KUKA KRL program: MyProgram_086().src

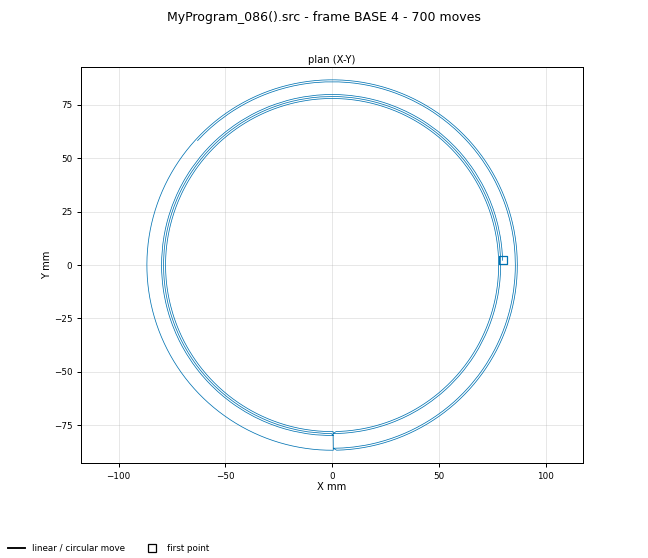
[picture p0: tool path of MyProgram_086().src in frame BASE 4, 700 of 700 moves have a stored position in this frame; points joined in program order, loops and branches not executed]
&ACCESS RVP
&REL 1
&PARAM TEMPLATE = C:\KRC\Roboter\Template\vorgabe
&PARAM EDITMASK = *
DEF MyProgram_086()
; ---- Setting reference (Base) ----
$BASE = BASE_DATA[4]

; --------------------------
; ---- Setting tool (TCP) ----
$TOOL = TOOL_DATA[3]
; --------------------------

$VEL.CP = VEL_APROX_PRINT
Startdeposition()
$VEL.CP = VEL_PRINT
LIN {X 79.8742,Y 2.2154,Z 84,A -3.1634,B 24.9021,C -2.2842,E1 25.1597,E2 447.7459} C_DIS
LIN {X 79.7565,Y 4.8855,Z 84,A -1.5386,B 24.9024,C -2.2808,E1 25.1594,E2 446.1387} C_DIS
LIN {X 79.546,Y 7.5648,Z 84,A 0.5064,B 24.9016,C -2.2907,E1 25.1589,E2 444.0824} C_DIS
LIN {X 79.2109,Y 10.5084,Z 84,A 2.7603,B 24.9006,C -2.3016,E1 25.1581,E2 441.8162} C_DIS
LIN {X 78.7938,Y 13.2771,Z 84,A 4.7205,B 24.9002,C -2.3063,E1 25.1573,E2 439.8564} C_DIS
LIN {X 77.6208,Y 18.9672,Z 84,A 8.4482,B 24.9003,C -2.305,E1 25.1551,E2 436.1534} C_DIS
LIN {X 76.3858,Y 23.452,Z 84,A 12.1024,B 24.8986,C -2.3252,E1 25.1523,E2 432.4725} C_DIS
LIN {X 75.4106,Y 26.4193,Z 84,A 14.3588,B 24.8979,C -2.3323,E1 25.1503,E2 430.2119} C_DIS
LIN {X 74.0231,Y 30.0886,Z 84,A 17.0668,B 24.8975,C -2.3371,E1 25.1475,E2 427.5076} C_DIS
LIN {X 72.6892,Y 33.1839,Z 84,A 19.5229,B 24.8968,C -2.3452,E1 25.1448,E2 425.0459} C_DIS
LIN {X 71.424,Y 35.8258,Z 84,A 21.7203,B 24.896,C -2.3541,E1 25.142,E2 422.8392} C_DIS
LIN {X 70.1389,Y 38.2794,Z 84,A 23.7,B 24.8956,C -2.3593,E1 25.1394,E2 420.8576} C_DIS
LIN {X 67.1297,Y 43.3403,Z 84,A 27.8834,B 24.8947,C -2.3691,E1 25.1333,E2 416.6724} C_DIS
LIN {X 65.2345,Y 46.1444,Z 84,A 30.2162,B 24.8944,C -2.3722,E1 25.1296,E2 414.3437} C_DIS
LIN {X 62.1422,Y 50.2304,Z 84,A 33.417,B 24.8949,C -2.3662,E1 25.1243,E2 411.1722} C_DIS
LIN {X 59.7766,Y 53.0248,Z 84,A 37.0655,B 24.8915,C -2.4041,E1 25.1174,E2 407.4506} C_DIS
LIN {X 57.5676,Y 55.4135,Z 84,A 39.0218,B 24.8921,C -2.3974,E1 25.1137,E2 405.5186} C_DIS
LIN {X 54.5308,Y 58.4041,Z 84,A 42.8995,B 24.8893,C -2.4292,E1 25.1057,E2 401.5814} C_DIS
LIN {X 50.973,Y 61.5346,Z 84,A 44.8682,B 24.8927,C -2.3915,E1 25.1017,E2 399.7098} C_DIS
LIN {X 49.2422,Y 62.9293,Z 84,A 46.8182,B 24.8914,C -2.4053,E1 25.0974,E2 397.7345} C_DIS
LIN {X 44.8304,Y 66.1436,Z 84,A 50.2204,B 24.8922,C -2.3963,E1 25.0898,E2 394.3654} C_DIS
LIN {X 42.7835,Y 67.4871,Z 84,A 52.2562,B 24.8912,C -2.4075,E1 25.085,E2 392.3098} C_DIS
LIN {X 40.8002,Y 68.703,Z 84,A 54.7814,B 24.8886,C -2.436,E1 25.0788,E2 389.7249} C_DIS
LIN {X 37.7018,Y 70.4522,Z 84,A 56.7061,B 24.8901,C -2.4204,E1 25.0741,E2 387.8427} C_DIS
LIN {X 34.3391,Y 72.1502,Z 84,A 59.5121,B 24.8895,C -2.4269,E1 25.0671,E2 385.0287} C_DIS
LIN {X 30.3149,Y 73.931,Z 84,A 62.4788,B 24.8897,C -2.4246,E1 25.0595,E2 382.0745} C_DIS
LIN {X 26.5785,Y 75.3548,Z 84,A 64.9595,B 24.8905,C -2.4159,E1 25.0531,E2 379.6198} C_DIS
LIN {X 24.1474,Y 76.17,Z 84,A 67.3413,B 24.8889,C -2.4333,E1 25.0467,E2 377.2012} C_DIS
LIN {X 21.1695,Y 77.05,Z 84,A 69.6421,B 24.8885,C -2.437,E1 25.0405,E2 374.8954} C_DIS
LIN {X 17.4919,Y 77.9679,Z 84,A 72.8738,B 24.887,C -2.4535,E1 25.0316,E2 371.6289} C_DIS
LIN {X 13.8906,Y 78.6883,Z 84,A 74.367,B 24.89,C -2.4213,E1 25.0277,E2 370.2138} C_DIS
LIN {X 8.6493,Y 79.4357,Z 84,A 78.2763,B 24.8896,C -2.4254,E1 25.0169,E2 366.2982} C_DIS
LIN {X 3.806,Y 79.8147,Z 84,A 82.6374,B 24.8873,C -2.4507,E1 25.0046,E2 361.8791} C_DIS
LIN {X 0.5734,Y 79.9025,Z 84,A 84.7785,B 24.8878,C -2.4452,E1 24.9986,E2 359.7512} C_DIS
LIN {X -3.1784,Y 79.8417,Z 84,A 87.9123,B 24.8867,C -2.457,E1 24.9898,E2 356.5887} C_DIS
LIN {X -7.2148,Y 79.5783,Z 84,A 89.9291,B 24.8891,C -2.4306,E1 24.9844,E2 354.6338} C_DIS
LIN {X -13.3811,Y 78.7764,Z 84,A 95.4024,B 24.8868,C -2.4562,E1 24.9691,E2 349.0949} C_DIS
LIN {X -17.7165,Y 77.9162,Z 84,A 97.6435,B 24.8894,C -2.4274,E1 24.9631,E2 346.9195} C_DIS
LIN {X -20.8905,Y 77.1254,Z 84,A 100.0246,B 24.8895,C -2.4261,E1 24.9567,E2 344.5381} C_DIS
LIN {X -26.7737,Y 75.2863,Z 84,A 104.5281,B 24.8898,C -2.4232,E1 24.9447,E2 340.0333} C_DIS
LIN {X -30.0238,Y 74.0495,Z 84,A 107.3916,B 24.8892,C -2.4299,E1 24.9372,E2 337.1475} C_DIS
LIN {X -34.5431,Y 72.0522,Z 84,A 110.4827,B 24.8908,C -2.4123,E1 24.9295,E2 334.0908} C_DIS
LIN {X -37.6093,Y 70.5015,Z 84,A 113.0625,B 24.8908,C -2.4113,E1 24.9231,E2 331.5062} C_DIS
LIN {X -42.7396,Y 67.5136,Z 84,A 117.0511,B 24.8922,C -2.3965,E1 24.9136,E2 327.5408} C_DIS
LIN {X -45.878,Y 65.421,Z 84,A 120.3122,B 24.8914,C -2.406,E1 24.906,E2 324.246} C_DIS
LIN {X -49.9813,Y 62.3441,Z 84,A 124.1225,B 24.8918,C -2.4017,E1 24.8976,E2 320.4319} C_DIS
LIN {X -52.7972,Y 59.9774,Z 84,A 126.8256,B 24.8921,C -2.3975,E1 24.8919,E2 317.7282} C_DIS
LIN {X -55.1723,Y 57.8006,Z 84,A 128.6467,B 24.8938,C -2.3792,E1 24.8883,E2 315.9432} C_DIS
LIN {X -57.5075,Y 55.4763,Z 84,A 131.6065,B 24.8929,C -2.3893,E1 24.8824,E2 312.9468} C_DIS
LIN {X -59.8884,Y 52.8992,Z 84,A 133.2739,B 24.8954,C -2.3607,E1 24.8795,E2 311.3401} C_DIS
LIN {X -61.9095,Y 50.5175,Z 84,A 135.7729,B 24.8954,C -2.3617,E1 24.875,E2 308.8273} C_DIS
LIN {X -65.6702,Y 45.5207,Z 84,A 140.2241,B 24.8965,C -2.3488,E1 24.8676,E2 304.3853} C_DIS
LIN {X -67.0145,Y 43.5198,Z 84,A 142.3289,B 24.896,C -2.3537,E1 24.8644,E2 302.2582} C_DIS
LIN {X -69.2019,Y 39.9481,Z 84,A 144.8295,B 24.8979,C -2.3322,E1 24.8608,E2 299.796} C_DIS
LIN {X -71.2813,Y 36.1081,Z 84,A 147.7071,B 24.8993,C -2.3167,E1 24.8571,E2 296.9403} C_DIS
LIN {X -72.814,Y 32.9069,Z 84,A 150.6411,B 24.8991,C -2.319,E1 24.8535,E2 293.9847} C_DIS
LIN {X -74.8991,Y 27.8408,Z 84,A 154.4993,B 24.9003,C -2.3053,E1 24.8495,E2 290.1378} C_DIS
LIN {X -76.4902,Y 23.1115,Z 84,A 158.2746,B 24.9008,C -2.2992,E1 24.8462,E2 286.3553} C_DIS
LIN {X -77.3182,Y 20.167,Z 84,A 160.5268,B 24.9013,C -2.2939,E1 24.8446,E2 284.1028} C_DIS
LIN {X -78.0736,Y 17.0075,Z 84,A 162.8457,B 24.9019,C -2.2863,E1 24.8431,E2 281.7885} C_DIS
LIN {X -78.7311,Y 13.6505,Z 84,A 166.1222,B 24.9008,C -2.2996,E1 24.8415,E2 278.4606} C_DIS
LIN {X -79.3072,Y 9.763,Z 84,A 168.4445,B 24.9027,C -2.2779,E1 24.8407,E2 276.1764} C_DIS
LIN {X -79.8336,Y 3.3663,Z 84,A 173.7794,B 24.9023,C -2.2821,E1 24.8398,E2 270.7993} C_DIS
LIN {X -79.8974,Y -1.1225,Z 84,A 175.7486,B 24.9059,C -2.2397,E1 24.8398,E2 268.9195} C_DIS
LIN {X -79.8317,Y -3.4108,Z 84,A 177.6251,B 24.9059,C -2.2405,E1 24.84,E2 267.0298} C_DIS
LIN {X -79.4763,Y -8.2616,Z 84,A -178.2229,B 24.9053,C -2.2466,E1 24.841,E2 262.8384} C_DIS
LIN {X -79.0723,Y -11.5061,Z 84,A -176.628,B 24.9076,C -2.22,E1 24.8416,E2 261.2975} C_DIS
LIN {X -78.6483,Y -14.113,Z 84,A -173.8348,B 24.9061,C -2.2373,E1 24.843,E2 258.4465} C_DIS
LIN {X -77.9265,Y -17.6722,Z 84,A -172.049,B 24.9085,C -2.2081,E1 24.844,E2 256.7197} C_DIS
LIN {X -77.2337,Y -20.4894,Z 84,A -169.8346,B 24.9088,C -2.2053,E1 24.8456,E2 254.4992} C_DIS
LIN {X -76.4721,Y -23.1726,Z 84,A -167.7993,B 24.9092,C -2.2002,E1 24.8472,E2 252.4643} C_DIS
LIN {X -75.6471,Y -25.7351,Z 84,A -165.9949,B 24.9099,C -2.1913,E1 24.8487,E2 250.6709} C_DIS
LIN {X -74.8294,Y -28.0247,Z 84,A -164.0957,B 24.91,C -2.1902,E1 24.8506,E2 248.7635} C_DIS
LIN {X -73.1802,Y -32.0845,Z 84,A -160.7297,B 24.9103,C -2.1871,E1 24.8542,E2 245.3863} C_DIS
LIN {X -71.665,Y -35.3396,Z 84,A -158.3657,B 24.9113,C -2.1744,E1 24.8571,E2 243.0397} C_DIS
LIN {X -70.2189,Y -38.132,Z 84,A -155.2566,B 24.91,C -2.1908,E1 24.8613,E2 239.8751} C_DIS
LIN {X -68.2289,Y -41.5881,Z 84,A -153.7955,B 24.9136,C -2.1466,E1 24.8632,E2 238.5119} C_DIS
LIN {X -65.3218,Y -46.022,Z 84,A -149.2606,B 24.9128,C -2.1561,E1 24.8703,E2 233.9316} C_DIS
LIN {X -63.2139,Y -48.8748,Z 84,A -146.7523,B 24.9134,C -2.149,E1 24.8745,E2 231.4282} C_DIS
LIN {X -61.0851,Y -51.5123,Z 84,A -143.5632,B 24.9122,C -2.1637,E1 24.8803,E2 228.1893} C_DIS
LIN {X -58.459,Y -54.474,Z 84,A -141.8,B 24.915,C -2.1287,E1 24.8835,E2 226.502} C_DIS
LIN {X -56.8071,Y -56.1934,Z 84,A -138.8409,B 24.9126,C -2.1587,E1 24.8895,E2 223.4585} C_DIS
LIN {X -53.5902,Y -59.2704,Z 84,A -136.8565,B 24.9157,C -2.1196,E1 24.8934,E2 221.5593} C_DIS
LIN {X -50.8929,Y -61.6012,Z 84,A -133.9567,B 24.9154,C -2.1241,E1 24.8996,E2 218.6378} C_DIS
LIN {X -47.3833,Y -64.3398,Z 84,A -131.2008,B 24.9168,C -2.1066,E1 24.9056,E2 215.9134} C_DIS
LIN {X -45.2583,Y -65.8529,Z 84,A -129.046,B 24.9164,C -2.1112,E1 24.9106,E2 213.7403} C_DIS
LIN {X -40.5803,Y -68.833,Z 84,A -125.0904,B 24.9169,C -2.1046,E1 24.92,E2 209.7878} C_DIS
LIN {X -36.4922,Y -71.085,Z 84,A -121.1636,B 24.916,C -2.1164,E1 24.9297,E2 205.8221} C_DIS
LIN {X -32.4299,Y -73.029,Z 84,A -117.9364,B 24.9163,C -2.1127,E1 24.9379,E2 202.5957} C_DIS
LIN {X -28.8497,Y -74.5157,Z 84,A -115.4468,B 24.9172,C -2.1018,E1 24.9443,E2 200.1266} C_DIS
LIN {X -25.242,Y -75.8134,Z 84,A -112.9215,B 24.9178,C -2.0932,E1 24.9509,E2 197.6168} C_DIS
LIN {X -22.0228,Y -76.8101,Z 84,A -110.403,B 24.9178,C -2.0944,E1 24.9577,E2 195.0912} C_DIS
LIN {X -18.1488,Y -77.8164,Z 84,A -107.4559,B 24.9177,C -2.095,E1 24.9657,E2 192.1384} C_DIS
LIN {X -11.9311,Y -79.0093,Z 84,A -103.2308,B 24.9185,C -2.0844,E1 24.9773,E2 187.9342} C_DIS
LIN {X -7.865,Y -79.5178,Z 84,A -100.2852,B 24.9185,C -2.0841,E1 24.9854,E2 184.9873} C_DIS
LIN {X -1.223,Y -79.8956,Z 84,A -95.4367,B 24.9183,C -2.0867,E1 24.9989,E2 180.1315} C_DIS
LIN {X 0.4916,Y -79.9011,Z 84,A -94.4036,B 24.9188,C -2.0813,E1 25.0018,E2 179.1113} C_DIS
Enddeposition()
LIN {X 0.4916,Y -79.9011,Z 84,A -94.4036,B 24.9188,C -2.0813,E1 25.0018,E2 179.1113} C_DIS
Startdeposition()
$VEL.CP = VEL_PRINT
LIN {X -0.3135,Y -78.968,Z 84,A -95.3503,B 24.9183,C -2.0869,E1 24.9992,E2 180.0445} C_DIS
LIN {X -3.6516,Y -78.8844,Z 84,A -98.627,B 24.9202,C -2.0625,E1 24.9899,E2 183.3797} C_DIS
LIN {X -11.2534,Y -78.1626,Z 84,A -103.0469,B 24.9177,C -2.0945,E1 24.9778,E2 187.7261} C_DIS
LIN {X -14.5877,Y -77.6101,Z 84,A -106.1891,B 24.9192,C -2.076,E1 24.969,E2 190.9155} C_DIS
LIN {X -16.7787,Y -77.1653,Z 84,A -108.0748,B 24.9197,C -2.0694,E1 24.9638,E2 192.819} C_DIS
LIN {X -20.6747,Y -76.214,Z 84,A -110.5178,B 24.9186,C -2.0839,E1 24.9573,E2 195.2311} C_DIS
LIN {X -22.947,Y -75.5622,Z 84,A -112.4428,B 24.9189,C -2.0793,E1 24.9521,E2 197.1703} C_DIS
LIN {X -25.8684,Y -74.6118,Z 84,A -114.6287,B 24.9187,C -2.0823,E1 24.9463,E2 199.3533} C_DIS
LIN {X -28.9712,Y -73.4622,Z 84,A -116.9095,B 24.9183,C -2.0878,E1 24.9404,E2 201.6258} C_DIS
LIN {X -32.0325,Y -72.1812,Z 84,A -119.3726,B 24.9182,C -2.0888,E1 24.9341,E2 204.0923} C_DIS
LIN {X -36.2142,Y -70.1757,Z 84,A -122.7661,B 24.9179,C -2.092,E1 24.9256,E2 207.4869} C_DIS
LIN {X -38.7437,Y -68.8114,Z 84,A -124.941,B 24.9179,C -2.0924,E1 24.9202,E2 209.667} C_DIS
LIN {X -41.5484,Y -67.1555,Z 84,A -126.977,B 24.9169,C -2.1046,E1 24.9154,E2 211.6804} C_DIS
LIN {X -43.8056,Y -65.7057,Z 84,A -129.2439,B 24.9174,C -2.0991,E1 24.9101,E2 213.9678} C_DIS
LIN {X -46.2466,Y -64.0116,Z 84,A -131.5956,B 24.9174,C -2.0975,E1 24.9047,E2 216.3313} C_DIS
LIN {X -49.3608,Y -61.642,Z 84,A -134.3541,B 24.9169,C -2.1047,E1 24.8986,E2 219.0829} C_DIS
LIN {X -51.9456,Y -59.4782,Z 84,A -136.6683,B 24.9163,C -2.1128,E1 24.8937,E2 221.3868} C_DIS
LIN {X -55.1934,Y -56.479,Z 84,A -139.9523,B 24.9159,C -2.1172,E1 24.8871,E2 224.6735} C_DIS
LIN {X -57.4405,Y -54.1905,Z 84,A -142.1633,B 24.9153,C -2.1252,E1 24.8828,E2 226.8751} C_DIS
LIN {X -59.8164,Y -51.5579,Z 84,A -144.8824,B 24.9151,C -2.1272,E1 24.8777,E2 229.6016} C_DIS
LIN {X -61.7506,Y -49.2238,Z 84,A -147.0713,B 24.9147,C -2.1326,E1 24.8739,E2 231.7878} C_DIS
LIN {X -63.6304,Y -46.7676,Z 84,A -149.2643,B 24.9142,C -2.1393,E1 24.8702,E2 233.9753} C_DIS
LIN {X -65.5292,Y -44.0681,Z 84,A -151.9051,B 24.9142,C -2.1391,E1 24.866,E2 236.6298} C_DIS
LIN {X -67.2981,Y -41.3171,Z 84,A -154.3464,B 24.9138,C -2.1435,E1 24.8624,E2 239.073} C_DIS
LIN {X -69.2715,Y -37.9152,Z 84,A -157.009,B 24.9128,C -2.1559,E1 24.8588,E2 241.72} C_DIS
LIN {X -70.7826,Y -35.012,Z 84,A -159.234,B 24.912,C -2.1662,E1 24.856,E2 243.9324} C_DIS
LIN {X -71.8479,Y -32.7722,Z 84,A -161.2121,B 24.912,C -2.1667,E1 24.8536,E2 245.92} C_DIS
LIN {X -73.5353,Y -28.7848,Z 84,A -164.4106,B 24.9113,C -2.1743,E1 24.8502,E2 249.1182} C_DIS
LIN {X -74.5845,Y -25.9463,Z 84,A -166.5469,B 24.9107,C -2.1822,E1 24.8482,E2 251.2478} C_DIS
LIN {X -75.5729,Y -22.9122,Z 84,A -168.9534,B 24.9103,C -2.1868,E1 24.8462,E2 253.6571} C_DIS
LIN {X -76.4644,Y -19.7285,Z 84,A -171.3517,B 24.9097,C -2.194,E1 24.8445,E2 256.052} C_DIS
LIN {X -77.032,Y -17.3852,Z 84,A -173.1734,B 24.9094,C -2.1976,E1 24.8433,E2 257.876} C_DIS
LIN {X -77.6747,Y -14.2379,Z 84,A -175.4862,B 24.9088,C -2.2052,E1 24.8421,E2 260.1842} C_DIS
LIN {X -78.2546,Y -10.6035,Z 84,A -178.1615,B 24.9081,C -2.2134,E1 24.841,E2 262.8559} C_DIS
LIN {X -78.6457,Y -7.1324,Z 84,A 179.4961,B 24.907,C -2.2261,E1 24.8403,E2 265.1819} C_DIS
LIN {X -78.8628,Y -4.0917,Z 84,A 177.1919,B 24.9066,C -2.2308,E1 24.8399,E2 267.4887} C_DIS
LIN {X -78.9651,Y -0.824,Z 84,A 174.8111,B 24.906,C -2.2381,E1 24.8398,E2 269.8665} C_DIS
LIN {X -78.9261,Y 2.5905,Z 84,A 172.4096,B 24.9052,C -2.2479,E1 24.8399,E2 272.259} C_DIS
LIN {X -78.6598,Y 6.9801,Z 84,A 169.0099,B 24.9048,C -2.2529,E1 24.8406,E2 275.6672} C_DIS
LIN {X -78.3239,Y 10.0692,Z 84,A 167.0162,B 24.9036,C -2.2665,E1 24.8412,E2 277.6404} C_DIS
LIN {X -77.8867,Y 13.026,Z 84,A 164.5681,B 24.9036,C -2.2665,E1 24.8422,E2 280.103} C_DIS
LIN {X -77.2923,Y 16.1864,Z 84,A 162.2629,B 24.9029,C -2.2746,E1 24.8435,E2 282.4026} C_DIS
LIN {X -76.618,Y 19.1276,Z 84,A 160.0282,B 24.9024,C -2.2804,E1 24.8449,E2 284.6366} C_DIS
LIN {X -75.8653,Y 21.9234,Z 84,A 157.8612,B 24.902,C -2.2853,E1 24.8466,E2 286.8045} C_DIS
LIN {X -75.0425,Y 24.5909,Z 84,A 155.6032,B 24.902,C -2.2859,E1 24.8485,E2 289.074} C_DIS
LIN {X -74.0216,Y 27.5146,Z 84,A 153.3477,B 24.9014,C -2.2925,E1 24.8507,E2 291.3264} C_DIS
LIN {X -72.6949,Y 30.8463,Z 84,A 151.0391,B 24.9001,C -2.3076,E1 24.8531,E2 293.6119} C_DIS
LIN {X -71.5223,Y 33.4752,Z 84,A 148.9221,B 24.8996,C -2.3131,E1 24.8556,E2 295.7273} C_DIS
LIN {X -70.2745,Y 36.021,Z 84,A 146.7527,B 24.8993,C -2.3164,E1 24.8583,E2 297.9005} C_DIS
LIN {X -68.1719,Y 39.859,Z 84,A 142.8838,B 24.9,C -2.3084,E1 24.8637,E2 301.8086} C_DIS
LIN {X -66.2415,Y 42.9911,Z 84,A 140.8879,B 24.8979,C -2.3324,E1 24.8666,E2 303.7573} C_DIS
LIN {X -63.7565,Y 46.5953,Z 84,A 137.3263,B 24.898,C -2.3315,E1 24.8724,E2 307.3386} C_DIS
LIN {X -61.1955,Y 49.9117,Z 84,A 134.8544,B 24.8961,C -2.3536,E1 24.8766,E2 309.7693} C_DIS
LIN {X -59.3682,Y 52.0716,Z 84,A 132.3649,B 24.8966,C -2.3479,E1 24.8812,E2 312.2837} C_DIS
LIN {X -56.6731,Y 54.993,Z 84,A 129.6752,B 24.8955,C -2.3598,E1 24.8863,E2 314.9567} C_DIS
LIN {X -54.3673,Y 57.2742,Z 84,A 127.3959,B 24.8948,C -2.3673,E1 24.8909,E2 317.2278} C_DIS
LIN {X -52.2189,Y 59.2396,Z 84,A 125.4995,B 24.8939,C -2.3776,E1 24.8948,E2 319.1072} C_DIS
LIN {X -50.0739,Y 61.0639,Z 84,A 123.0109,B 24.8945,C -2.3707,E1 24.9002,E2 321.6217} C_DIS
LIN {X -47.3137,Y 63.2253,Z 84,A 120.4553,B 24.8941,C -2.3757,E1 24.9058,E2 324.1746} C_DIS
LIN {X -43.7728,Y 65.7273,Z 84,A 117.6723,B 24.8927,C -2.3912,E1 24.9121,E2 326.9301} C_DIS
LIN {X -41.9961,Y 66.8755,Z 84,A 115.8451,B 24.8931,C -2.3866,E1 24.9165,E2 328.7742} C_DIS
LIN {X -39.1445,Y 68.584,Z 84,A 113.6552,B 24.8922,C -2.3966,E1 24.9217,E2 330.9469} C_DIS
LIN {X -36.3929,Y 70.0841,Z 84,A 111.0691,B 24.8926,C -2.3923,E1 24.9281,E2 333.5505} C_DIS
LIN {X -33.2515,Y 71.6265,Z 84,A 108.7755,B 24.8917,C -2.4026,E1 24.9339,E2 335.8253} C_DIS
LIN {X -30.9833,Y 72.6372,Z 84,A 106.8361,B 24.8917,C -2.4016,E1 24.9388,E2 337.7716} C_DIS
LIN {X -28.0442,Y 73.821,Z 84,A 104.5278,B 24.8915,C -2.4045,E1 24.9448,E2 340.0781} C_DIS
LIN {X -23.7017,Y 75.3282,Z 84,A 101.3146,B 24.8908,C -2.4117,E1 24.9533,E2 343.2802} C_DIS
LIN {X -21.3793,Y 76.0195,Z 84,A 99.5364,B 24.8908,C -2.413,E1 24.9581,E2 345.0581} C_DIS
LIN {X -18.6628,Y 76.7314,Z 84,A 97.5178,B 24.8905,C -2.4155,E1 24.9635,E2 347.0737} C_DIS
LIN {X -15.2375,Y 77.485,Z 84,A 94.6051,B 24.8912,C -2.4078,E1 24.9716,E2 350.0082} C_DIS
LIN {X -9.5718,Y 78.3869,Z 84,A 90.7353,B 24.8902,C -2.4184,E1 24.9822,E2 353.8559} C_DIS
LIN {X -5.4515,Y 78.7801,Z 84,A 87.2166,B 24.8914,C -2.4058,E1 24.9921,E2 357.4063} C_DIS
LIN {X 1.31,Y 78.9577,Z 84,A 82.7899,B 24.8901,C -2.4202,E1 25.0043,E2 361.799} C_DIS
LIN {X 4.1367,Y 78.8603,Z 84,A 80.2315,B 24.8913,C -2.4063,E1 25.0116,E2 364.3896} C_DIS
LIN {X 8.9308,Y 78.4622,Z 84,A 77.2015,B 24.8902,C -2.4187,E1 25.0199,E2 367.3884} C_DIS
LIN {X 12.1275,Y 78.0316,Z 84,A 74.8413,B 24.8903,C -2.4175,E1 25.0264,E2 369.7491} C_DIS
LIN {X 16.3395,Y 77.2609,Z 84,A 71.7711,B 24.8903,C -2.4172,E1 25.0348,E2 372.8164} C_DIS
LIN {X 18.9682,Y 76.6569,Z 84,A 69.9746,B 24.89,C -2.4207,E1 25.0397,E2 374.6021} C_DIS
LIN {X 21.5611,Y 75.968,Z 84,A 67.8747,B 24.8905,C -2.4151,E1 25.0454,E2 376.712} C_DIS
LIN {X 24.6184,Y 75.0337,Z 84,A 65.4826,B 24.8909,C -2.4112,E1 25.0517,E2 379.1088} C_DIS
LIN {X 26.8794,Y 74.2532,Z 84,A 63.8944,B 24.8906,C -2.4139,E1 25.0559,E2 380.6874} C_DIS
LIN {X 29.5861,Y 73.2169,Z 84,A 61.0395,B 24.8928,C -2.3903,E1 25.0634,E2 383.5919} C_DIS
LIN {X 32.9059,Y 71.7873,Z 84,A 58.8986,B 24.8918,C -2.4011,E1 25.0688,E2 385.7018} C_DIS
LIN {X 36.3828,Y 70.0893,Z 84,A 56.1972,B 24.8918,C -2.4006,E1 25.0755,E2 388.3969} C_DIS
LIN {X 40.1048,Y 68.0266,Z 84,A 53.2732,B 24.8918,C -2.4011,E1 25.0826,E2 391.3111} C_DIS
LIN {X 42.6665,Y 66.4498,Z 84,A 51.0113,B 24.8923,C -2.3955,E1 25.0879,E2 393.5792} C_DIS
LIN {X 45.8019,Y 64.3289,Z 84,A 48.4166,B 24.8923,C -2.3955,E1 25.0939,E2 396.165} C_DIS
LIN {X 47.877,Y 62.8008,Z 84,A 46.399,B 24.893,C -2.3877,E1 25.0984,E2 398.1936} C_DIS
LIN {X 50.7877,Y 60.4714,Z 84,A 42.8215,B 24.8958,C -2.3569,E1 25.1062,E2 401.8304} C_DIS
LIN {X 53.9952,Y 57.6242,Z 84,A 40.6692,B 24.8938,C -2.3791,E1 25.1105,E2 403.9213} C_DIS
LIN {X 55.5586,Y 56.1182,Z 84,A 38.5346,B 24.8956,C -2.3591,E1 25.1148,E2 406.0943} C_DIS
LIN {X 57.8314,Y 53.7748,Z 84,A 36.6711,B 24.8947,C -2.369,E1 25.1183,E2 407.9262} C_DIS
LIN {X 59.9681,Y 51.3798,Z 84,A 34.425,B 24.8949,C -2.3663,E1 25.1225,E2 410.1688} C_DIS
LIN {X 62.0163,Y 48.8876,Z 84,A 32.4349,B 24.8945,C -2.3714,E1 25.1259,E2 412.1374} C_DIS
LIN {X 63.5074,Y 46.9355,Z 84,A 30.2999,B 24.8958,C -2.3563,E1 25.1295,E2 414.2979} C_DIS
LIN {X 65.1196,Y 44.673,Z 84,A 28.1998,B 24.8965,C -2.3487,E1 25.1329,E2 416.4057} C_DIS
LIN {X 69.0588,Y 38.3007,Z 84,A 23.1976,B 24.8965,C -2.3478,E1 25.1401,E2 421.3845} C_DIS
LIN {X 70.347,Y 35.8791,Z 84,A 20.8554,B 24.898,C -2.3315,E1 25.1432,E2 423.7527} C_DIS
LIN {X 71.8446,Y 32.7794,Z 84,A 18.4041,B 24.8985,C -2.326,E1 25.1461,E2 426.204} C_DIS
LIN {X 73.0589,Y 29.9741,Z 84,A 16.1398,B 24.8992,C -2.3182,E1 25.1486,E2 428.4743} C_DIS
LIN {X 74.3098,Y 26.7244,Z 84,A 13.7732,B 24.8994,C -2.3158,E1 25.1509,E2 430.8333} C_DIS
LIN {X 75.2667,Y 23.8981,Z 84,A 11.6324,B 24.8999,C -2.3101,E1 25.1527,E2 432.9754} C_DIS
LIN {X 76.2159,Y 20.6676,Z 84,A 9.1974,B 24.9005,C -2.303,E1 25.1546,E2 435.4132} C_DIS
LIN {X 76.7171,Y 18.7213,Z 84,A 7.3399,B 24.9019,C -2.2862,E1 25.1558,E2 437.2997} C_DIS
LIN {X 77.7416,Y 13.866,Z 84,A 4.3396,B 24.9013,C -2.2938,E1 25.1575,E2 440.2647} C_DIS
LIN {X 78.1513,Y 11.3327,Z 84,A 2.2765,B 24.9023,C -2.2817,E1 25.1583,E2 442.3442} C_DIS
LIN {X 78.5612,Y 8.0123,Z 84,A -0.1762,B 24.9031,C -2.2732,E1 25.1591,E2 444.8023} C_DIS
LIN {X 78.8299,Y 4.6861,Z 84,A -2.2311,B 24.9027,C -2.2771,E1 25.1595,E2 446.8359} C_DIS
LIN {X 78.9356,Y 2.2812,Z 84,A -4.2791,B 24.904,C -2.2621,E1 25.1598,E2 448.9072} C_DIS
LIN {X 78.9622,Y -1.0615,Z 84,A -6.6901,B 24.9046,C -2.2548,E1 25.1598,E2 451.321} C_DIS
LIN {X 78.8519,Y -4.2878,Z 84,A -8.9354,B 24.905,C -2.2503,E1 25.1595,E2 453.5635} C_DIS
LIN {X 78.6569,Y -7.0119,Z 84,A -10.9987,B 24.9058,C -2.2414,E1 25.159,E2 455.6356} C_DIS
LIN {X 78.3684,Y -9.7253,Z 84,A -13.0089,B 24.9064,C -2.2341,E1 25.1583,E2 457.6511} C_DIS
LIN {X 77.7196,Y -13.9881,Z 84,A -16.3854,B 24.9078,C -2.2165,E1 25.1568,E2 461.0495} C_DIS
LIN {X 76.8423,Y -18.2063,Z 84,A -18.9453,B 24.9072,C -2.2243,E1 25.1553,E2 463.576} C_DIS
LIN {X 75.9811,Y -21.5147,Z 84,A -21.5819,B 24.9082,C -2.2116,E1 25.1534,E2 466.2274} C_DIS
LIN {X 75.0766,Y -24.4858,Z 84,A -23.7984,B 24.9087,C -2.2058,E1 25.1515,E2 468.4451} C_DIS
LIN {X 74.091,Y -27.3241,Z 84,A -25.9872,B 24.9093,C -2.1988,E1 25.1495,E2 470.6381} C_DIS
LIN {X 73.006,Y -30.103,Z 84,A -28.09,B 24.9097,C -2.1941,E1 25.1473,E2 472.7403} C_DIS
LIN {X 71.7055,Y -33.0796,Z 84,A -30.8027,B 24.9112,C -2.176,E1 25.1441,E2 475.4811} C_DIS
LIN {X 68.7473,Y -38.8586,Z 84,A -35.3236,B 24.9118,C -2.1681,E1 25.1382,E2 479.9969} C_DIS
LIN {X 66.7188,Y -42.2475,Z 84,A -38.0788,B 24.9122,C -2.1634,E1 25.1342,E2 482.7492} C_DIS
LIN {X 65.1173,Y -44.6763,Z 84,A -40.5082,B 24.9135,C -2.1477,E1 25.1304,E2 485.2035} C_DIS
LIN {X 61.8719,Y -49.0703,Z 84,A -44.3206,B 24.914,C -2.1418,E1 25.1239,E2 489.0118} C_DIS
LIN {X 59.2159,Y -52.246,Z 84,A -47.0533,B 24.914,C -2.1424,E1 25.119,E2 491.7307} C_DIS
LIN {X 55.3644,Y -56.31,Z 84,A -50.9085,B 24.9142,C -2.1388,E1 25.1115,E2 495.5777} C_DIS
LIN {X 53.3675,Y -58.2058,Z 84,A -53.0691,B 24.915,C -2.1291,E1 25.1071,E2 497.7523} C_DIS
LIN {X 50.8358,Y -60.4314,Z 84,A -55.3177,B 24.915,C -2.1296,E1 25.1024,E2 499.991} C_DIS
LIN {X 46.534,Y -63.8014,Z 84,A -59.9076,B 24.9171,C -2.1023,E1 25.0921,E2 504.6288} C_DIS
LIN {X 42.971,Y -66.2544,Z 84,A -62.5984,B 24.9165,C -2.1096,E1 25.0859,E2 507.2934} C_DIS
LIN {X 40.1912,Y -67.9756,Z 84,A -64.8082,B 24.9165,C -2.1101,E1 25.0806,E2 509.495} C_DIS
LIN {X 36.4357,Y -70.0615,Z 84,A -68.8046,B 24.919,C -2.0785,E1 25.0707,E2 513.5547} C_DIS
LIN {X 33.0997,Y -71.6971,Z 84,A -70.5806,B 24.9172,C -2.1016,E1 25.0663,E2 515.2716} C_DIS
LIN {X 29.4775,Y -73.2611,Z 84,A -73.5936,B 24.9179,C -2.0929,E1 25.0585,E2 518.2979} C_DIS
LIN {X 26.7558,Y -74.2983,Z 84,A -75.735,B 24.9181,C -2.0893,E1 25.0529,E2 520.4434} C_DIS
LIN {X 23.8875,Y -75.2701,Z 84,A -77.8635,B 24.9181,C -2.0887,E1 25.0473,E2 522.5694} C_DIS
LIN {X 19.4927,Y -76.525,Z 84,A -81.182,B 24.9185,C -2.0851,E1 25.0383,E2 525.891} C_DIS
LIN {X 16.3993,Y -77.2481,Z 84,A -83.5962,B 24.9189,C -2.0797,E1 25.0317,E2 528.3146} C_DIS
LIN {X 13.0847,Y -77.8768,Z 84,A -85.8211,B 24.9185,C -2.0843,E1 25.0257,E2 530.5262} C_DIS
LIN {X 8.977,Y -78.4568,Z 84,A -88.9358,B 24.9189,C -2.0793,E1 25.017,E2 533.6503} C_DIS
LIN {X 5.8883,Y -78.7496,Z 84,A -91.3432,B 24.9194,C -2.0737,E1 25.0103,E2 536.0696} C_DIS
LIN {X 2.8532,Y -78.918,Z 84,A -93.4393,B 24.9192,C -2.076,E1 25.0044,E2 538.1596} C_DIS
LIN {X 0.4855,Y -78.9628,Z 84,A -94.5822,B 24.9179,C -2.092,E1 25.0014,E2 539.2643} C_DIS
Enddeposition()
LIN {X 0.4855,Y -78.9628,Z 84,A -94.5822,B 24.9179,C -2.092,E1 25.0014,E2 539.2643} C_DIS
Startdeposition()
$VEL.CP = VEL_PRINT
LIN {X 1.9087,Y -78.0103,Z 84,A -93.2608,B 24.916,C -2.1164,E1 25.0052,E2 537.8853} C_DIS
LIN {X 3.8193,Y -77.9401,Z 84,A -91.599,B 24.9154,C -2.1243,E1 25.0099,E2 536.2052} C_DIS
LIN {X 6.6951,Y -77.746,Z 84,A -89.4717,B 24.9153,C -2.1257,E1 25.0158,E2 534.0758} C_DIS
LIN {X 9.5849,Y -77.4426,Z 84,A -87.6166,B 24.9158,C -2.1189,E1 25.0209,E2 532.2382} C_DIS
LIN {X 11.4698,Y -77.1861,Z 84,A -86.2209,B 24.9158,C -2.1198,E1 25.0248,E2 530.8415} C_DIS
LIN {X 13.3494,Y -76.8833,Z 84,A -84.5762,B 24.9151,C -2.128,E1 25.0294,E2 529.179} C_DIS
LIN {X 16.1545,Y -76.3432,Z 84,A -82.4734,B 24.9149,C -2.13,E1 25.0351,E2 527.0741} C_DIS
LIN {X 18.8089,Y -75.7322,Z 84,A -80.7203,B 24.9153,C -2.1247,E1 25.0398,E2 525.3361} C_DIS
LIN {X 20.7756,Y -75.217,Z 84,A -79.1902,B 24.9151,C -2.1274,E1 25.044,E2 523.8021} C_DIS
LIN {X 23.3767,Y -74.4489,Z 84,A -77.2336,B 24.9151,C -2.1286,E1 25.0492,E2 521.8459} C_DIS
LIN {X 25.3808,Y -73.7907,Z 84,A -75.7127,B 24.9149,C -2.1297,E1 25.0532,E2 520.3255} C_DIS
LIN {X 27.3039,Y -73.1003,Z 84,A -73.9769,B 24.9142,C -2.1387,E1 25.0578,E2 518.572} C_DIS
LIN {X 30.3075,Y -71.9061,Z 84,A -71.7398,B 24.9142,C -2.138,E1 25.0636,E2 516.3417} C_DIS
LIN {X 32.6099,Y -70.8925,Z 84,A -69.7729,B 24.9138,C -2.1444,E1 25.0686,E2 514.3646} C_DIS
LIN {X 34.985,Y -69.7511,Z 84,A -68.0757,B 24.9141,C -2.1404,E1 25.0728,E2 512.6814} C_DIS
LIN {X 36.8481,Y -68.7853,Z 84,A -66.2968,B 24.9133,C -2.1501,E1 25.0773,E2 510.8844} C_DIS
LIN {X 39.1967,Y -67.4743,Z 84,A -64.5716,B 24.9136,C -2.1461,E1 25.0814,E2 509.1739} C_DIS
LIN {X 41.2957,Y -66.2095,Z 84,A -62.6564,B 24.9131,C -2.153,E1 25.086,E2 507.2485} C_DIS
LIN {X 43.3507,Y -64.8843,Z 84,A -60.8662,B 24.9128,C -2.1563,E1 25.0902,E2 505.4563} C_DIS
LIN {X 45.6074,Y -63.3176,Z 84,A -58.9808,B 24.9128,C -2.1563,E1 25.0945,E2 503.5773} C_DIS
LIN {X 47.6145,Y -61.8215,Z 84,A -57.0617,B 24.9123,C -2.1627,E1 25.0988,E2 501.6501} C_DIS
LIN {X 49.8326,Y -60.0479,Z 84,A -54.9567,B 24.9118,C -2.1679,E1 25.1033,E2 499.5409} C_DIS
LIN {X 51.9943,Y -58.1862,Z 84,A -52.8656,B 24.9115,C -2.1726,E1 25.1077,E2 497.447} C_DIS
LIN {X 54.2099,Y -56.1278,Z 84,A -50.5485,B 24.9108,C -2.1808,E1 25.1124,E2 495.12} C_DIS
LIN {X 56.6146,Y -53.7022,Z 84,A -48.1336,B 24.9105,C -2.184,E1 25.1171,E2 492.7078} C_DIS
LIN {X 58.4559,Y -51.693,Z 84,A -46.1122,B 24.9101,C -2.1897,E1 25.1209,E2 490.6821} C_DIS
LIN {X 60.2722,Y -49.5627,Z 84,A -44.0377,B 24.9096,C -2.1956,E1 25.1246,E2 488.6031} C_DIS
LIN {X 62.1704,Y -47.1593,Z 84,A -41.7901,B 24.9091,C -2.2016,E1 25.1285,E2 486.3521} C_DIS
LIN {X 63.7681,Y -44.976,Z 84,A -40.054,B 24.9093,C -2.1992,E1 25.1313,E2 484.63} C_DIS
LIN {X 64.881,Y -43.3557,Z 84,A -38.442,B 24.9085,C -2.2084,E1 25.1338,E2 483.0041} C_DIS
LIN {X 66.3664,Y -41.0445,Z 84,A -36.6037,B 24.9085,C -2.2085,E1 25.1365,E2 481.1749} C_DIS
LIN {X 67.8273,Y -38.5824,Z 84,A -34.5142,B 24.908,C -2.2142,E1 25.1395,E2 479.0829} C_DIS
LIN {X 68.8915,Y -36.6484,Z 84,A -32.6881,B 24.9071,C -2.2253,E1 25.1419,E2 477.2399} C_DIS
LIN {X 70.1801,Y -34.1161,Z 84,A -30.6065,B 24.9066,C -2.2313,E1 25.1445,E2 475.1553} C_DIS
LIN {X 71.3221,Y -31.6604,Z 84,A -28.8205,B 24.9066,C -2.2309,E1 25.1466,E2 473.38} C_DIS
LIN {X 72.3707,Y -29.1819,Z 84,A -26.889,B 24.9063,C -2.2355,E1 25.1486,E2 471.4482} C_DIS
LIN {X 73.3126,Y -26.7262,Z 84,A -24.8819,B 24.9056,C -2.2438,E1 25.1506,E2 469.4326} C_DIS
LIN {X 74.3475,Y -23.698,Z 84,A -22.6407,B 24.9052,C -2.2477,E1 25.1526,E2 467.195} C_DIS
LIN {X 74.9792,Y -21.6167,Z 84,A -20.8313,B 24.9042,C -2.2593,E1 25.154,E2 465.3685} C_DIS
LIN {X 75.6644,Y -19.0804,Z 84,A -19.0612,B 24.9042,C -2.2604,E1 25.1553,E2 463.606} C_DIS
LIN {X 76.3107,Y -16.3038,Z 84,A -17.0719,B 24.9039,C -2.2637,E1 25.1565,E2 461.6204} C_DIS
LIN {X 76.7331,Y -14.1847,Z 84,A -15.2529,B 24.9028,C -2.2761,E1 25.1574,E2 459.7829} C_DIS
LIN {X 77.1597,Y -11.64,Z 84,A -13.6164,B 24.903,C -2.274,E1 25.1582,E2 458.161} C_DIS
LIN {X 77.418,Y -9.7751,Z 84,A -12.2484,B 24.9026,C -2.278,E1 25.1587,E2 456.7917} C_DIS
LIN {X 77.6577,Y -7.6515,Z 84,A -10.5989,B 24.902,C -2.2855,E1 25.1591,E2 455.1341} C_DIS
LIN {X 77.8784,Y -4.9099,Z 84,A -8.6652,B 24.9017,C -2.2892,E1 25.1595,E2 453.203} C_DIS
LIN {X 78.0005,Y -2.2322,Z 84,A -6.6888,B 24.9011,C -2.2958,E1 25.1597,E2 451.2229} C_DIS
LIN {X 78.0303,Y 0.5696,Z 84,A -4.6033,B 24.9005,C -2.3032,E1 25.1597,E2 449.1322} C_DIS
LIN {X 77.9485,Y 3.6238,Z 84,A -2.4231,B 24.9,C -2.3084,E1 25.1596,E2 446.9529} C_DIS
LIN {X 77.8218,Y 5.7462,Z 84,A -0.9072,B 24.8997,C -2.3119,E1 25.1593,E2 445.4377} C_DIS
LIN {X 77.5719,Y 8.471,Z 84,A 1.1028,B 24.8992,C -2.3183,E1 25.1587,E2 443.4246} C_DIS
LIN {X 77.324,Y 10.5005,Z 84,A 2.7305,B 24.8984,C -2.3269,E1 25.1581,E2 441.786} C_DIS
LIN {X 76.8733,Y 13.4054,Z 84,A 4.9975,B 24.8975,C -2.337,E1 25.1571,E2 439.5084} C_DIS
LIN {X 76.2311,Y 16.6689,Z 84,A 7.2503,B 24.8974,C -2.3386,E1 25.1558,E2 437.265} C_DIS
LIN {X 75.7263,Y 18.8331,Z 84,A 8.7835,B 24.8972,C -2.3405,E1 25.1548,E2 435.7361} C_DIS
LIN {X 75.2094,Y 20.8039,Z 84,A 10.4529,B 24.8963,C -2.3505,E1 25.1536,E2 434.0529} C_DIS
LIN {X 74.4286,Y 23.442,Z 84,A 12.2767,B 24.8963,C -2.3504,E1 25.1521,E2 432.2397} C_DIS
LIN {X 73.7902,Y 25.3824,Z 84,A 13.7557,B 24.896,C -2.3541,E1 25.1508,E2 430.7601} C_DIS
LIN {X 73.1,Y 27.3048,Z 84,A 15.4844,B 24.895,C -2.3657,E1 25.1491,E2 429.0139} C_DIS
LIN {X 72.0994,Y 29.8483,Z 84,A 17.2389,B 24.8952,C -2.3636,E1 25.1473,E2 427.274} C_DIS
LIN {X 71.3386,Y 31.6238,Z 84,A 18.649,B 24.8948,C -2.3674,E1 25.1457,E2 425.8627} C_DIS
LIN {X 70.5423,Y 33.3624,Z 84,A 20.0452,B 24.8945,C -2.371,E1 25.1441,E2 424.4653} C_DIS
LIN {X 69.7035,Y 35.081,Z 84,A 21.4409,B 24.8942,C -2.3747,E1 25.1423,E2 423.0685} C_DIS
LIN {X 68.7515,Y 36.9104,Z 84,A 23.175,B 24.8932,C -2.3856,E1 25.14,E2 421.3178} C_DIS
LIN {X 67.369,Y 39.3776,Z 84,A 25.251,B 24.8927,C -2.3911,E1 25.1371,E2 419.2395} C_DIS
LIN {X 65.9744,Y 41.6721,Z 84,A 27.0539,B 24.8927,C -2.3911,E1 25.1345,E2 417.4459} C_DIS
LIN {X 64.4322,Y 44.0185,Z 84,A 29.0232,B 24.8925,C -2.3934,E1 25.1315,E2 415.4807} C_DIS
LIN {X 63.243,Y 45.712,Z 84,A 30.7794,B 24.8915,C -2.4044,E1 25.1286,E2 413.707} C_DIS
LIN {X 61.5513,Y 47.965,Z 84,A 32.8151,B 24.8912,C -2.4084,E1 25.1251,E2 411.6716} C_DIS
LIN {X 59.7507,Y 50.1903,Z 84,A 34.8828,B 24.8908,C -2.4122,E1 25.1214,E2 409.6043} C_DIS
LIN {X 57.8694,Y 52.3481,Z 84,A 36.9723,B 24.8904,C -2.4166,E1 25.1176,E2 407.5139} C_DIS
LIN {X 55.911,Y 54.4348,Z 84,A 39.0705,B 24.89,C -2.421,E1 25.1135,E2 405.4143} C_DIS
LIN {X 53.8598,Y 56.4652,Z 84,A 41.1722,B 24.8896,C -2.4249,E1 25.1093,E2 403.3122} C_DIS
LIN {X 51.7117,Y 58.4392,Z 84,A 43.293,B 24.8893,C -2.4285,E1 25.1049,E2 401.1913} C_DIS
LIN {X 49.5538,Y 60.2795,Z 84,A 45.404,B 24.8889,C -2.4333,E1 25.1003,E2 399.0771} C_DIS
LIN {X 47.1511,Y 62.1766,Z 84,A 47.6572,B 24.8885,C -2.4375,E1 25.0954,E2 396.8223} C_DIS
LIN {X 44.9997,Y 63.7512,Z 84,A 49.3721,B 24.8889,C -2.4336,E1 25.0915,E2 395.1226} C_DIS
LIN {X 42.9261,Y 65.1643,Z 84,A 51.264,B 24.8884,C -2.438,E1 25.0871,E2 393.2265} C_DIS
LIN {X 41.0469,Y 66.3649,Z 84,A 52.8471,B 24.8884,C -2.4389,E1 25.0834,E2 391.6464} C_DIS
LIN {X 38.5636,Y 67.8381,Z 84,A 54.9641,B 24.8881,C -2.4418,E1 25.0783,E2 389.5288} C_DIS
LIN {X 36.6663,Y 68.882,Z 84,A 56.7706,B 24.8873,C -2.4503,E1 25.0738,E2 387.7075} C_DIS
LIN {X 34.3592,Y 70.0613,Z 84,A 58.444,B 24.8877,C -2.446,E1 25.0697,E2 386.0488} C_DIS
LIN {X 32.4041,Y 70.987,Z 84,A 60.2611,B 24.8869,C -2.4545,E1 25.065,E2 384.2162} C_DIS
LIN {X 29.915,Y 72.0715,Z 84,A 62.1654,B 24.8869,C -2.454,E1 25.0601,E2 382.3175} C_DIS
LIN {X 27.3174,Y 73.0952,Z 84,A 64.0524,B 24.8872,C -2.4513,E1 25.0552,E2 380.4411} C_DIS
LIN {X 25.3819,Y 73.7904,Z 84,A 65.5561,B 24.8872,C -2.4524,E1 25.0513,E2 378.9378} C_DIS
LIN {X 22.6538,Y 74.6731,Z 84,A 67.6602,B 24.887,C -2.454,E1 25.0457,E2 376.8338} C_DIS
LIN {X 20.8178,Y 75.2055,Z 84,A 69.0608,B 24.8869,C -2.4549,E1 25.0419,E2 375.4335} C_DIS
LIN {X 18.533,Y 75.7995,Z 84,A 70.9172,B 24.8865,C -2.4594,E1 25.0369,E2 373.569} C_DIS
LIN {X 16.2976,Y 76.3121,Z 84,A 72.7111,B 24.8861,C -2.4633,E1 25.032,E2 371.7682} C_DIS
LIN {X 13.3391,Y 76.8852,Z 84,A 74.9363,B 24.8861,C -2.4645,E1 25.0258,E2 369.5426} C_DIS
LIN {X 10.6475,Y 77.3031,Z 84,A 76.6841,B 24.8866,C -2.458,E1 25.0211,E2 367.812} C_DIS
LIN {X 8.7597,Y 77.5397,Z 84,A 78.0938,B 24.8866,C -2.4586,E1 25.0171,E2 366.4019} C_DIS
LIN {X 6.6098,Y 77.7528,Z 84,A 79.9161,B 24.8859,C -2.4653,E1 25.012,E2 364.5646} C_DIS
LIN {X 4.0092,Y 77.9298,Z 84,A 81.678,B 24.8863,C -2.4611,E1 25.0072,E2 362.8135} C_DIS
LIN {X 1.1049,Y 78.0251,Z 84,A 83.7271,B 24.8866,C -2.4585,E1 25.0015,E2 360.7709} C_DIS
LIN {X -1.0593,Y 78.026,Z 84,A 85.5513,B 24.886,C -2.4646,E1 24.9963,E2 358.9321} C_DIS
LIN {X -3.6836,Y 77.946,Z 84,A 87.3132,B 24.8865,C -2.4594,E1 24.9914,E2 357.1822} C_DIS
LIN {X -6.516,Y 77.7603,Z 84,A 89.5532,B 24.8862,C -2.4628,E1 24.9852,E2 354.9332} C_DIS
LIN {X -9.4019,Y 77.4645,Z 84,A 91.4654,B 24.8868,C -2.4557,E1 24.9799,E2 353.0368} C_DIS
LIN {X -11.5324,Y 77.1764,Z 84,A 93.3072,B 24.8862,C -2.4618,E1 24.9748,E2 351.1788} C_DIS
LIN {X -14.9497,Y 76.5871,Z 84,A 95.598,B 24.8871,C -2.453,E1 24.9685,E2 348.9067} C_DIS
LIN {X -17.5384,Y 76.0358,Z 84,A 97.6291,B 24.8871,C -2.4537,E1 24.963,E2 346.8715} C_DIS
LIN {X -19.8807,Y 75.4587,Z 84,A 99.3085,B 24.8874,C -2.4494,E1 24.9585,E2 345.1997} C_DIS
LIN {X -21.7206,Y 74.9497,Z 84,A 100.9865,B 24.8868,C -2.4554,E1 24.9539,E2 343.505} C_DIS
LIN {X -24.579,Y 74.0611,Z 84,A 103.1614,B 24.8871,C -2.4522,E1 24.9481,E2 341.3336} C_DIS
LIN {X -27.1858,Y 73.145,Z 84,A 104.9507,B 24.888,C -2.4433,E1 24.9435,E2 339.562} C_DIS
LIN {X -28.8469,Y 72.5052,Z 84,A 106.2836,B 24.888,C -2.4422,E1 24.94,E2 338.2287} C_DIS
LIN {X -30.8762,Y 71.6645,Z 84,A 108.1148,B 24.8877,C -2.4457,E1 24.9353,E2 336.385} C_DIS
LIN {X -33.3657,Y 70.5407,Z 84,A 110.1539,B 24.8879,C -2.4435,E1 24.9301,E2 334.346} C_DIS
LIN {X -35.9315,Y 69.2689,Z 84,A 112.0772,B 24.8887,C -2.4354,E1 24.9254,E2 332.4369} C_DIS
LIN {X -38.3331,Y 67.9685,Z 84,A 114.0981,B 24.889,C -2.4324,E1 24.9204,E2 330.4173} C_DIS
LIN {X -40.7991,Y 66.5174,Z 84,A 116.1378,B 24.8895,C -2.427,E1 24.9156,E2 328.3841} C_DIS
LIN {X -42.6653,Y 65.3362,Z 84,A 117.9874,B 24.8892,C -2.4299,E1 24.9112,E2 326.5218} C_DIS
LIN {X -44.79,Y 63.8982,Z 84,A 119.704,B 24.8899,C -2.4218,E1 24.9073,E2 324.8186} C_DIS
LIN {X -47.0548,Y 62.249,Z 84,A 121.7264,B 24.8904,C -2.4167,E1 24.9027,E2 322.8012} C_DIS
LIN {X -49.1907,Y 60.5748,Z 84,A 123.8307,B 24.8905,C -2.4153,E1 24.8981,E2 320.6924} C_DIS
LIN {X -51.1618,Y 58.9199,Z 84,A 125.81,B 24.8907,C -2.4134,E1 24.8939,E2 318.7099} C_DIS
LIN {X -53.4152,Y 56.8845,Z 84,A 127.9784,B 24.8913,C -2.4068,E1 24.8895,E2 316.5487} C_DIS
LIN {X -55.4667,Y 54.886,Z 84,A 130.0945,B 24.8917,C -2.4021,E1 24.8853,E2 314.4347} C_DIS
LIN {X -57.4434,Y 52.8138,Z 84,A 132.222,B 24.8921,C -2.3976,E1 24.8812,E2 312.3087} C_DIS
LIN {X -59.3614,Y 50.6484,Z 84,A 134.3428,B 24.8926,C -2.3921,E1 24.8774,E2 310.1914} C_DIS
LIN {X -61.222,Y 48.3828,Z 84,A 136.5951,B 24.8929,C -2.389,E1 24.8734,E2 307.936} C_DIS
LIN {X -63.1841,Y 45.7925,Z 84,A 138.8058,B 24.8939,C -2.3782,E1 24.8697,E2 305.7404} C_DIS
LIN {X -64.3523,Y 44.1365,Z 84,A 140.2775,B 24.8943,C -2.3737,E1 24.8674,E2 304.2721} C_DIS
LIN {X -65.7651,Y 42.0002,Z 84,A 142.2888,B 24.8944,C -2.3718,E1 24.8643,E2 302.2553} C_DIS
LIN {X -67.3298,Y 39.4439,Z 84,A 144.3879,B 24.8952,C -2.363,E1 24.8613,E2 300.1663} C_DIS
LIN {X -68.3279,Y 37.6894,Z 84,A 145.9039,B 24.8955,C -2.3596,E1 24.8593,E2 298.6505} C_DIS
LIN {X -69.545,Y 35.3912,Z 84,A 147.8465,B 24.8959,C -2.3549,E1 24.8568,E2 296.7088} C_DIS
LIN {X -70.5402,Y 33.3667,Z 84,A 149.4706,B 24.8964,C -2.3492,E1 24.8548,E2 295.0896} C_DIS
LIN {X -71.3358,Y 31.6301,Z 84,A 150.8818,B 24.8968,C -2.3452,E1 24.8532,E2 293.6801} C_DIS
LIN {X -72.0885,Y 29.8748,Z 84,A 152.366,B 24.897,C -2.343,E1 24.8516,E2 292.1929} C_DIS
LIN {X -73.0893,Y 27.3331,Z 84,A 154.4208,B 24.8974,C -2.3381,E1 24.8495,E2 290.1382} C_DIS
LIN {X -74.0583,Y 24.5873,Z 84,A 156.5633,B 24.898,C -2.3317,E1 24.8476,E2 287.999} C_DIS
LIN {X -74.9109,Y 21.8522,Z 84,A 158.5997,B 24.8987,C -2.3235,E1 24.8459,E2 285.9704} C_DIS
LIN {X -75.6627,Y 19.0869,Z 84,A 160.6953,B 24.8993,C -2.3167,E1 24.8444,E2 283.8788} C_DIS
LIN {X -76.137,Y 17.0999,Z 84,A 162.2141,B 24.8997,C -2.3124,E1 24.8435,E2 282.3613} C_DIS
LIN {X -76.737,Y 14.1629,Z 84,A 164.6737,B 24.8997,C -2.3119,E1 24.8421,E2 279.8885} C_DIS
LIN {X -77.1908,Y 11.438,Z 84,A 166.7163,B 24.9002,C -2.3058,E1 24.8413,E2 277.8483} C_DIS
LIN {X -77.5425,Y 8.7359,Z 84,A 168.5003,B 24.9013,C -2.2941,E1 24.8407,E2 276.0816} C_DIS
LIN {X -77.7553,Y 6.5791,Z 84,A 170.3352,B 24.9012,C -2.295,E1 24.8402,E2 274.2334} C_DIS
LIN {X -77.9306,Y 3.994,Z 84,A 172.025,B 24.9022,C -2.2837,E1 24.8399,E2 272.5605} C_DIS
LIN {X -78.01,Y 1.9219,Z 84,A 173.5414,B 24.9026,C -2.2787,E1 24.8399,E2 271.0469} C_DIS
LIN {X -78.0302,Y -0.5779,Z 84,A 175.4694,B 24.9029,C -2.2751,E1 24.8399,E2 269.1158} C_DIS
LIN {X -77.9566,Y -3.4365,Z 84,A 177.6567,B 24.9033,C -2.2707,E1 24.84,E2 266.926} C_DIS
LIN {X -77.7577,Y -6.5484,Z 84,A 179.8109,B 24.9042,C -2.2601,E1 24.8404,E2 264.7842} C_DIS
LIN {X -77.5744,Y -8.4468,Z 84,A -178.766,B 24.9045,C -2.2562,E1 24.8408,E2 263.3617} C_DIS
LIN {X -77.323,Y -10.5074,Z 84,A -177.0295,B 24.9045,C -2.2567,E1 24.8415,E2 261.6137} C_DIS
LIN {X -76.8856,Y -13.3363,Z 84,A -175.1273,B 24.9054,C -2.2452,E1 24.8423,E2 259.7276} C_DIS
LIN {X -76.3448,Y -16.1469,Z 84,A -172.7772,B 24.9054,C -2.2449,E1 24.8436,E2 257.3643} C_DIS
LIN {X -75.7273,Y -18.829,Z 84,A -170.9616,B 24.9064,C -2.2337,E1 24.8448,E2 255.5649} C_DIS
LIN {X -75.2063,Y -20.8153,Z 84,A -169.46,B 24.9068,C -2.229,E1 24.8459,E2 254.0658} C_DIS
LIN {X -74.6736,Y -22.6519,Z 84,A -168.0445,B 24.9071,C -2.2251,E1 24.847,E2 252.6515} C_DIS
LIN {X -74.0962,Y -24.4748,Z 84,A -166.6312,B 24.9075,C -2.2211,E1 24.8482,E2 251.2395} C_DIS
LIN {X -73.2696,Y -26.8442,Z 84,A -164.7019,B 24.9077,C -2.2179,E1 24.85,E2 249.3069} C_DIS
LIN {X -72.493,Y -28.878,Z 84,A -163.1442,B 24.9082,C -2.2123,E1 24.8516,E2 247.7539} C_DIS
LIN {X -71.6611,Y -30.8841,Z 84,A -161.3297,B 24.9082,C -2.2133,E1 24.8536,E2 245.927} C_DIS
LIN {X -70.5378,Y -33.3717,Z 84,A -159.3009,B 24.9085,C -2.2083,E1 24.856,E2 243.8991} C_DIS
LIN {X -69.2665,Y -35.9361,Z 84,A -157.3539,B 24.9093,C -2.1986,E1 24.8585,E2 241.9647} C_DIS
LIN {X -67.9664,Y -38.3368,Z 84,A -155.4026,B 24.9099,C -2.1919,E1 24.8611,E2 240.0191} C_DIS
LIN {X -66.9419,Y -40.1002,Z 84,A -153.6405,B 24.9097,C -2.1947,E1 24.8636,E2 238.2413} C_DIS
LIN {X -65.3275,Y -42.6786,Z 84,A -151.4279,B 24.9102,C -2.1885,E1 24.8669,E2 236.0324} C_DIS
LIN {X -63.8688,Y -44.8323,Z 84,A -149.7413,B 24.911,C -2.178,E1 24.8696,E2 234.3624} C_DIS
LIN {X -62.674,Y -46.489,Z 84,A -148.0143,B 24.9108,C -2.1801,E1 24.8725,E2 232.622} C_DIS
LIN {X -60.9654,Y -48.7075,Z 84,A -145.9393,B 24.9112,C -2.1758,E1 24.876,E2 230.5476} C_DIS
LIN {X -59.0928,Y -50.9636,Z 84,A -143.7993,B 24.9116,C -2.1705,E1 24.8799,E2 228.4104} C_DIS
LIN {X -57.1694,Y -53.1124,Z 84,A -141.6555,B 24.912,C -2.1665,E1 24.8839,E2 226.2665} C_DIS
LIN {X -55.1829,Y -55.1734,Z 84,A -139.544,B 24.9123,C -2.1623,E1 24.8881,E2 224.156} C_DIS
LIN {X -53.1226,Y -57.1598,Z 84,A -137.4283,B 24.9126,C -2.1585,E1 24.8924,E2 222.0408} C_DIS
LIN {X -51.0775,Y -58.9935,Z 84,A -135.387,B 24.9129,C -2.1552,E1 24.8967,E2 219.9992} C_DIS
LIN {X -48.8175,Y -60.8773,Z 84,A -133.2308,B 24.9132,C -2.1511,E1 24.9013,E2 217.8446} C_DIS
LIN {X -46.497,Y -62.668,Z 84,A -131.072,B 24.9135,C -2.1476,E1 24.9061,E2 215.6865} C_DIS
LIN {X -44.144,Y -64.3472,Z 84,A -129.0871,B 24.9141,C -2.1404,E1 24.9106,E2 213.7119} C_DIS
LIN {X -41.8459,Y -65.8641,Z 84,A -127.1363,B 24.9145,C -2.1354,E1 24.9152,E2 211.7667} C_DIS
LIN {X -39.6419,Y -67.2128,Z 84,A -125.172,B 24.9145,C -2.1345,E1 24.9199,E2 209.7986} C_DIS
LIN {X -37.6336,Y -68.3591,Z 84,A -123.4563,B 24.9147,C -2.1326,E1 24.9241,E2 208.0823} C_DIS
LIN {X -35.2224,Y -69.6313,Z 84,A -121.4435,B 24.9149,C -2.1304,E1 24.9291,E2 206.0693} C_DIS
LIN {X -32.6522,Y -70.8728,Z 84,A -119.3362,B 24.915,C -2.1283,E1 24.9344,E2 203.9617} C_DIS
LIN {X -30.0218,Y -72.0265,Z 84,A -117.3011,B 24.9154,C -2.1241,E1 24.9396,E2 201.9319} C_DIS
LIN {X -28.0808,Y -72.8061,Z 84,A -115.7697,B 24.9155,C -2.1225,E1 24.9436,E2 200.4009} C_DIS
LIN {X -25.3871,Y -73.7886,Z 84,A -113.6582,B 24.9156,C -2.1208,E1 24.9491,E2 198.2891} C_DIS
LIN {X -22.6591,Y -74.6714,Z 84,A -111.4535,B 24.9156,C -2.122,E1 24.955,E2 196.0777} C_DIS
LIN {X -20.0204,Y -75.421,Z 84,A -109.5322,B 24.9159,C -2.1182,E1 24.9602,E2 194.1625} C_DIS
LIN {X -17.8871,Y -75.9552,Z 84,A -107.6836,B 24.9154,C -2.1238,E1 24.9652,E2 192.298} C_DIS
LIN {X -15.3589,Y -76.5065,Z 84,A -105.9326,B 24.9158,C -2.1189,E1 24.97,E2 190.5568} C_DIS
LIN {X -12.556,Y -77.0161,Z 84,A -103.9213,B 24.916,C -2.116,E1 24.9755,E2 188.5504} C_DIS
LIN {X -10.6817,Y -77.2983,Z 84,A -102.5293,B 24.916,C -2.1157,E1 24.9794,E2 187.1579} C_DIS
LIN {X -8.8086,Y -77.5339,Z 84,A -101.126,B 24.916,C -2.1159,E1 24.9833,E2 185.7531} C_DIS
LIN {X -6.5629,Y -77.7565,Z 84,A -99.249,B 24.9155,C -2.122,E1 24.9885,E2 183.8606} C_DIS
LIN {X -3.9913,Y -77.9307,Z 84,A -97.5789,B 24.916,C -2.1158,E1 24.9931,E2 182.2048} C_DIS
LIN {X -1.9744,Y -78.0084,Z 84,A -95.9053,B 24.9156,C -2.1215,E1 24.9979,E2 180.5175} C_DIS
LIN {X 0.4843,Y -78.0291,Z 84,A -94.9006,B 24.9174,C -2.0992,E1 25.0005,E2 179.5658} C_DIS
Enddeposition()
LIN {X 0.5852,Y -86.7766,Z 85,A -93.8702,B 24.9262,C -1.9835,E1 25.0026,E2 178.8098} C_DIS
Startdeposition()
$VEL.CP = VEL_PRINT
LIN {X -2.6891,Y -86.7371,Z 85,A -96.8683,B 24.9282,C -1.9565,E1 24.9941,E2 181.8722} C_DIS
LIN {X -5.8798,Y -86.5794,Z 85,A -98.9773,B 24.9282,C -1.9564,E1 24.9882,E2 183.9821} C_DIS
LIN {X -9.0626,Y -86.3043,Z 85,A -101.087,B 24.9282,C -1.9565,E1 24.9823,E2 186.0926} C_DIS
LIN {X -12.1097,Y -85.9298,Z 85,A -103.159,B 24.9283,C -1.9555,E1 24.9766,E2 188.1685} C_DIS
LIN {X -15.3335,Y -85.4134,Z 85,A -105.2908,B 24.9283,C -1.9569,E1 24.9707,E2 190.2991} C_DIS
LIN {X -18.4669,Y -84.7911,Z 85,A -107.4021,B 24.9281,C -1.9577,E1 24.9649,E2 192.4109} C_DIS
LIN {X -21.5753,Y -84.0539,Z 85,A -109.5138,B 24.9281,C -1.9588,E1 24.9592,E2 194.5231} C_DIS
LIN {X -24.6545,Y -83.2029,Z 85,A -111.6263,B 24.928,C -1.9601,E1 24.9535,E2 196.6359} C_DIS
LIN {X -27.7003,Y -82.239,Z 85,A -113.7393,B 24.9279,C -1.9616,E1 24.9479,E2 198.7491} C_DIS
LIN {X -30.7593,Y -81.1445,Z 85,A -115.8701,B 24.9277,C -1.9639,E1 24.9423,E2 200.8787} C_DIS
LIN {X -33.6751,Y -79.9784,Z 85,A -117.967,B 24.9276,C -1.9653,E1 24.9369,E2 202.9771} C_DIS
LIN {X -36.596,Y -78.6848,Z 85,A -120.0814,B 24.9274,C -1.9675,E1 24.9315,E2 205.0914} C_DIS
LIN {X -39.4674,Y -77.2844,Z 85,A -122.1965,B 24.9272,C -1.9698,E1 24.9263,E2 207.2065} C_DIS
LIN {X -42.2853,Y -75.7794,Z 85,A -124.3121,B 24.9271,C -1.9725,E1 24.9211,E2 209.3219} C_DIS
LIN {X -45.0923,Y -74.1434,Z 85,A -126.4455,B 24.9268,C -1.9759,E1 24.9159,E2 211.4536} C_DIS
LIN {X -47.7454,Y -72.4634,Z 85,A -128.5446,B 24.9266,C -1.9783,E1 24.911,E2 213.5537} C_DIS
LIN {X -50.3802,Y -70.6569,Z 85,A -130.6618,B 24.9264,C -1.9815,E1 24.9062,E2 215.6704} C_DIS
LIN {X -52.9468,Y -68.7546,Z 85,A -132.7793,B 24.9261,C -1.985,E1 24.9014,E2 217.7873} C_DIS
LIN {X -55.4416,Y -66.7592,Z 85,A -134.8973,B 24.9259,C -1.9886,E1 24.8969,E2 219.9046} C_DIS
LIN {X -57.8612,Y -64.6733,Z 85,A -137.0157,B 24.9256,C -1.9924,E1 24.8924,E2 222.0223} C_DIS
LIN {X -60.2024,Y -62.4998,Z 85,A -139.1346,B 24.9253,C -1.9964,E1 24.8881,E2 224.1404} C_DIS
LIN {X -62.4998,Y -60.2024,Z 85,A -141.2713,B 24.9249,C -2.0012,E1 24.8839,E2 226.2748} C_DIS
LIN {X -64.6733,Y -57.8612,Z 85,A -143.3909,B 24.9246,C -2.0056,E1 24.8799,E2 228.3934} C_DIS
LIN {X -66.7592,Y -55.4416,Z 85,A -145.5111,B 24.9242,C -2.0101,E1 24.8761,E2 230.5126} C_DIS
LIN {X -68.7546,Y -52.9468,Z 85,A -147.6315,B 24.9239,C -2.0147,E1 24.8724,E2 232.6318} C_DIS
LIN {X -70.6569,Y -50.3802,Z 85,A -149.7523,B 24.9235,C -2.0196,E1 24.869,E2 234.7514} C_DIS
LIN {X -72.44,Y -47.7809,Z 85,A -151.8599,B 24.9232,C -2.0241,E1 24.8657,E2 236.8587} C_DIS
LIN {X -74.1434,Y -45.0923,Z 85,A -153.9775,B 24.9228,C -2.0291,E1 24.8625,E2 238.9753} C_DIS
LIN {X -75.7794,Y -42.2853,Z 85,A -156.1109,B 24.9223,C -2.0351,E1 24.8596,E2 241.1053} C_DIS
LIN {X -77.2844,Y -39.4674,Z 85,A -158.2391,B 24.9219,C -2.0403,E1 24.8568,E2 243.2324} C_DIS
LIN {X -78.6848,Y -36.596,Z 85,A -160.3614,B 24.9215,C -2.0458,E1 24.8543,E2 245.3531} C_DIS
LIN {X -79.9784,Y -33.6751,Z 85,A -162.4842,B 24.9211,C -2.0514,E1 24.8519,E2 247.4742} C_DIS
LIN {X -81.1445,Y -30.7593,Z 85,A -164.5896,B 24.9207,C -2.0565,E1 24.8498,E2 249.5793} C_DIS
LIN {X -82.239,Y -27.7003,Z 85,A -166.7301,B 24.9202,C -2.063,E1 24.8478,E2 251.7166} C_DIS
LIN {X -83.2029,Y -24.6545,Z 85,A -168.8536,B 24.9197,C -2.0689,E1 24.8461,E2 253.8382} C_DIS
LIN {X -84.0539,Y -21.5753,Z 85,A -170.9772,B 24.9193,C -2.0749,E1 24.8445,E2 255.9599} C_DIS
LIN {X -84.7911,Y -18.4669,Z 85,A -173.101,B 24.9188,C -2.0809,E1 24.8432,E2 258.0817} C_DIS
LIN {X -85.4134,Y -15.3335,Z 85,A -175.2249,B 24.9183,C -2.087,E1 24.8421,E2 260.2036} C_DIS
LIN {X -85.9122,Y -12.2331,Z 85,A -177.3315,B 24.9179,C -2.0926,E1 24.8412,E2 262.3095} C_DIS
LIN {X -86.3043,Y -9.0626,Z 85,A -179.4556,B 24.9174,C -2.0988,E1 24.8405,E2 264.4315} C_DIS
LIN {X -86.5794,Y -5.8798,Z 85,A 178.4201,B 24.9169,C -2.105,E1 24.8401,E2 266.5535} C_DIS
LIN {X -86.7371,Y -2.6891,Z 85,A 176.2959,B 24.9164,C -2.1113,E1 24.8398,E2 268.6756} C_DIS
LIN {X -86.7792,Y 0.3519,Z 85,A 174.1868,B 24.9161,C -2.1149,E1 24.8398,E2 270.7888} C_DIS
LIN {X -86.6976,Y 3.7533,Z 85,A 172.0298,B 24.9153,C -2.1246,E1 24.84,E2 272.9357} C_DIS
LIN {X -86.505,Y 6.8877,Z 85,A 169.9228,B 24.9149,C -2.1303,E1 24.8404,E2 275.0418} C_DIS
LIN {X -86.1929,Y 10.067,Z 85,A 167.7982,B 24.9144,C -2.1366,E1 24.841,E2 277.1641} C_DIS
LIN {X -85.764,Y 13.2327,Z 85,A 165.674,B 24.9139,C -2.1429,E1 24.8419,E2 279.2858} C_DIS
LIN {X -85.2085,Y 16.4338,Z 85,A 163.5322,B 24.9133,C -2.1498,E1 24.8429,E2 281.4239} C_DIS
LIN {X -84.5581,Y 19.506,Z 85,A 161.4254,B 24.9129,C -2.1554,E1 24.8442,E2 283.5296} C_DIS
LIN {X -83.7829,Y 22.6052,Z 85,A 159.3014,B 24.9124,C -2.1616,E1 24.8457,E2 285.6512} C_DIS
LIN {X -82.8941,Y 25.6737,Z 85,A 157.1774,B 24.9119,C -2.1678,E1 24.8474,E2 287.7727} C_DIS
LIN {X -81.8749,Y 28.7587,Z 85,A 155.0361,B 24.9113,C -2.1745,E1 24.8493,E2 289.9102} C_DIS
LIN {X -80.7808,Y 31.7022,Z 85,A 152.9298,B 24.9109,C -2.18,E1 24.8514,E2 292.0154} C_DIS
LIN {X -79.5375,Y 34.7038,Z 85,A 150.7888,B 24.9103,C -2.1865,E1 24.8537,E2 294.1525} C_DIS
LIN {X -78.2062,Y 37.6079,Z 85,A 148.6655,B 24.9098,C -2.1924,E1 24.8562,E2 296.2733} C_DIS
LIN {X -76.8056,Y 40.3914,Z 85,A 146.5672,B 24.9094,C -2.1973,E1 24.8589,E2 298.3712} C_DIS
LIN {X -75.2277,Y 43.2592,Z 85,A 144.4195,B 24.9089,C -2.2039,E1 24.8618,E2 300.5144} C_DIS
LIN {X -73.6133,Y 45.9527,Z 85,A 142.3142,B 24.9085,C -2.2089,E1 24.8649,E2 302.6187} C_DIS
LIN {X -71.9212,Y 48.5583,Z 85,A 140.2179,B 24.9081,C -2.2133,E1 24.8681,E2 304.7149} C_DIS
LIN {X -70.0333,Y 51.2435,Z 85,A 138.0698,B 24.9076,C -2.2197,E1 24.8716,E2 306.8583} C_DIS
LIN {X -68.0997,Y 53.7865,Z 85,A 135.9481,B 24.9071,C -2.2249,E1 24.8752,E2 308.9776} C_DIS
LIN {X -66.0386,Y 56.298,Z 85,A 133.8092,B 24.9067,C -2.2306,E1 24.879,E2 311.1127} C_DIS
LIN {X -63.9584,Y 58.6505,Z 85,A 131.7054,B 24.9063,C -2.235,E1 24.883,E2 313.2155} C_DIS
LIN {X -61.7563,Y 60.9649,Z 85,A 129.5847,B 24.9059,C -2.2398,E1 24.8871,E2 315.3339} C_DIS
LIN {X -59.4309,Y 63.2339,Z 85,A 127.4469,B 24.9054,C -2.245,E1 24.8914,E2 317.468} C_DIS
LIN {X -57.0632,Y 65.3785,Z 85,A 125.3268,B 24.9051,C -2.2495,E1 24.8958,E2 319.5859} C_DIS
LIN {X -54.6181,Y 67.4346,Z 85,A 123.2072,B 24.9047,C -2.2538,E1 24.9003,E2 321.7033} C_DIS
LIN {X -52.1425,Y 69.3666,Z 85,A 121.1055,B 24.9044,C -2.2574,E1 24.905,E2 323.8042} C_DIS
LIN {X -49.554,Y 71.2388,Z 85,A 118.9868,B 24.9041,C -2.2613,E1 24.9098,E2 325.9208} C_DIS
LIN {X -46.8526,Y 73.0438,Z 85,A 116.851,B 24.9037,C -2.2657,E1 24.9148,E2 328.0531} C_DIS
LIN {X -44.1791,Y 74.6912,Z 85,A 114.7505,B 24.9034,C -2.2687,E1 24.9198,E2 330.153} C_DIS
LIN {X -41.4,Y 76.2667,Z 85,A 112.6329,B 24.9032,C -2.2721,E1 24.925,E2 332.2687} C_DIS
LIN {X -38.516,Y 77.7629,Z 85,A 110.4985,B 24.9028,C -2.2759,E1 24.9303,E2 334.3997} C_DIS
LIN {X -35.6773,Y 79.1056,Z 85,A 108.3995,B 24.9026,C -2.2783,E1 24.9356,E2 336.4982} C_DIS
LIN {X -32.7414,Y 80.3652,Z 85,A 106.2834,B 24.9024,C -2.2811,E1 24.941,E2 338.6126} C_DIS
LIN {X -29.7612,Y 81.5158,Z 85,A 104.168,B 24.9022,C -2.2836,E1 24.9465,E2 340.7263} C_DIS
LIN {X -26.7407,Y 82.556,Z 85,A 102.0531,B 24.902,C -2.286,E1 24.9521,E2 342.8396} C_DIS
LIN {X -23.7377,Y 83.4691,Z 85,A 99.9554,B 24.9018,C -2.2875,E1 24.9578,E2 344.9371} C_DIS
LIN {X -20.595,Y 84.2995,Z 85,A 97.8247,B 24.9016,C -2.2901,E1 24.9635,E2 347.0648} C_DIS
LIN {X -17.4782,Y 85.0004,Z 85,A 95.7112,B 24.9015,C -2.2918,E1 24.9693,E2 349.1769} C_DIS
LIN {X -14.3378,Y 85.5862,Z 85,A 93.5983,B 24.9013,C -2.2932,E1 24.9751,E2 351.2885} C_DIS
LIN {X -11.1779,Y 86.0559,Z 85,A 91.4859,B 24.9013,C -2.2945,E1 24.9809,E2 353.3995} C_DIS
LIN {X -8.0028,Y 86.409,Z 85,A 89.3741,B 24.9011,C -2.2955,E1 24.9868,E2 355.5101} C_DIS
LIN {X -4.7626,Y 86.648,Z 85,A 87.2456,B 24.9011,C -2.2969,E1 24.9927,E2 357.6361} C_DIS
LIN {X -1.5701,Y 86.7646,Z 85,A 85.1348,B 24.901,C -2.2974,E1 24.9986,E2 359.7458} C_DIS
LIN {X 1.5701,Y 86.7646,Z 85,A 83.0421,B 24.901,C -2.2972,E1 25.0044,E2 361.839} C_DIS
LIN {X 4.7626,Y 86.648,Z 85,A 80.9323,B 24.901,C -2.2972,E1 25.0103,E2 363.9479} C_DIS
LIN {X 8.0028,Y 86.409,Z 85,A 78.8073,B 24.901,C -2.2978,E1 25.0162,E2 366.0707} C_DIS
LIN {X 11.1779,Y 86.0559,Z 85,A 76.6974,B 24.901,C -2.2974,E1 25.0221,E2 368.1799} C_DIS
LIN {X 14.3378,Y 85.5862,Z 85,A 74.5897,B 24.901,C -2.2968,E1 25.0279,E2 370.287} C_DIS
LIN {X 17.4782,Y 85.0004,Z 85,A 72.4822,B 24.9011,C -2.296,E1 25.0337,E2 372.394} C_DIS
LIN {X 20.5422,Y 84.3124,Z 85,A 70.3925,B 24.9012,C -2.2943,E1 25.0394,E2 374.4846} C_DIS
LIN {X 23.6839,Y 83.4843,Z 85,A 68.2689,B 24.9013,C -2.2936,E1 25.0451,E2 376.6064} C_DIS
LIN {X 26.6922,Y 82.5717,Z 85,A 66.1795,B 24.9015,C -2.2916,E1 25.0506,E2 378.6969} C_DIS
LIN {X 29.7612,Y 81.5158,Z 85,A 64.0577,B 24.9015,C -2.2904,E1 25.0562,E2 380.8172} C_DIS
LIN {X 32.7414,Y 80.3652,Z 85,A 61.953,B 24.9017,C -2.2885,E1 25.0617,E2 382.9218} C_DIS
LIN {X 35.6773,Y 79.1056,Z 85,A 59.8488,B 24.9019,C -2.2863,E1 25.0671,E2 385.026} C_DIS
LIN {X 38.516,Y 77.7629,Z 85,A 57.7624,B 24.9022,C -2.2834,E1 25.0723,E2 387.1138} C_DIS
LIN {X 41.4,Y 76.2667,Z 85,A 55.6419,B 24.9024,C -2.2813,E1 25.0776,E2 389.2332} C_DIS
LIN {X 44.1791,Y 74.6912,Z 85,A 53.5392,B 24.9026,C -2.2786,E1 25.0826,E2 391.3361} C_DIS
LIN {X 46.8526,Y 73.0438,Z 85,A 51.4543,B 24.9029,C -2.275,E1 25.0876,E2 393.4228} C_DIS
LIN {X 49.5094,Y 71.2698,Z 85,A 49.3525,B 24.9032,C -2.2718,E1 25.0924,E2 395.525} C_DIS
LIN {X 52.1425,Y 69.3666,Z 85,A 47.2337,B 24.9034,C -2.269,E1 25.0972,E2 397.643} C_DIS
LIN {X 54.6181,Y 67.4346,Z 85,A 45.1502,B 24.9038,C -2.2648,E1 25.1018,E2 399.7285} C_DIS
LIN {X 57.1041,Y 65.3428,Z 85,A 43.0325,B 24.904,C -2.2616,E1 25.1063,E2 401.8456} C_DIS
LIN {X 59.4705,Y 63.1966,Z 85,A 40.9324,B 24.9044,C -2.2577,E1 25.1106,E2 403.9465} C_DIS
LIN {X 61.7563,Y 60.9649,Z 85,A 38.8329,B 24.9047,C -2.2536,E1 25.1147,E2 406.0469} C_DIS
LIN {X 63.9584,Y 58.6505,Z 85,A 36.7336,B 24.9051,C -2.2493,E1 25.1187,E2 408.1471} C_DIS
LIN {X 66.0386,Y 56.298,Z 85,A 34.6521,B 24.9055,C -2.2443,E1 25.1226,E2 410.231} C_DIS
LIN {X 68.0997,Y 53.7865,Z 85,A 32.5366,B 24.9059,C -2.2402,E1 25.1263,E2 412.3464} C_DIS
LIN {X 70.0333,Y 51.2435,Z 85,A 30.4445,B 24.9062,C -2.2357,E1 25.1298,E2 414.4392} C_DIS
LIN {X 71.8415,Y 48.676,Z 85,A 28.3579,B 24.9067,C -2.23,E1 25.1331,E2 416.5289} C_DIS
LIN {X 73.6133,Y 45.9527,Z 85,A 26.2434,B 24.9071,C -2.2255,E1 25.1363,E2 418.6434} C_DIS
LIN {X 75.2277,Y 43.2592,Z 85,A 24.1632,B 24.9076,C -2.2198,E1 25.1392,E2 420.7264} C_DIS
LIN {X 76.7943,Y 40.4128,Z 85,A 22.0494,B 24.908,C -2.215,E1 25.142,E2 422.8403} C_DIS
LIN {X 78.2297,Y 37.5589,Z 85,A 19.9529,B 24.9084,C -2.2096,E1 25.1446,E2 424.9385} C_DIS
LIN {X 79.5375,Y 34.7038,Z 85,A 17.8737,B 24.9089,C -2.2035,E1 25.147,E2 427.0207} C_DIS
LIN {X 80.7808,Y 31.7022,Z 85,A 15.7606,B 24.9093,C -2.1985,E1 25.1492,E2 429.1341} C_DIS
LIN {X 81.8929,Y 28.7074,Z 85,A 13.6648,B 24.9098,C -2.1927,E1 25.1512,E2 431.2317} C_DIS
LIN {X 82.878,Y 25.7256,Z 85,A 11.5864,B 24.9103,C -2.1864,E1 25.153,E2 433.3134} C_DIS
LIN {X 83.7829,Y 22.6052,Z 85,A 9.4738,B 24.9108,C -2.181,E1 25.1546,E2 435.4265} C_DIS
LIN {X 84.5581,Y 19.506,Z 85,A 7.3785,B 24.9113,C -2.1751,E1 25.156,E2 437.5237} C_DIS
LIN {X 85.2085,Y 16.4338,Z 85,A 5.3007,B 24.9118,C -2.1685,E1 25.1571,E2 439.6048} C_DIS
LIN {X 85.764,Y 13.2327,Z 85,A 3.1886,B 24.9123,C -2.1629,E1 25.1581,E2 441.7177} C_DIS
LIN {X 86.1929,Y 10.067,Z 85,A 1.0937,B 24.9128,C -2.1568,E1 25.1588,E2 443.8147} C_DIS
LIN {X 86.505,Y 6.8877,Z 85,A -0.9988,B 24.9132,C -2.1507,E1 25.1594,E2 445.9092} C_DIS
LIN {X 86.6976,Y 3.7533,Z 85,A -3.0783,B 24.9138,C -2.1439,E1 25.1597,E2 447.9923} C_DIS
LIN {X 86.7792,Y 0.3519,Z 85,A -5.2807,B 24.9142,C -2.1382,E1 25.1597,E2 450.195} C_DIS
LIN {X 86.7216,Y -3.1941,Z 85,A -7.7258,B 24.9151,C -2.1272,E1 25.1597,E2 452.6518} C_DIS
LIN {X 86.5453,Y -6.384,Z 85,A -9.835,B 24.9157,C -2.1204,E1 25.1592,E2 454.7644} C_DIS
LIN {X 86.2517,Y -9.5651,Z 85,A -11.9296,B 24.9162,C -2.1141,E1 25.1586,E2 456.8614} C_DIS
LIN {X 85.8412,Y -12.7333,Z 85,A -14.0241,B 24.9167,C -2.1079,E1 25.1578,E2 458.9583} C_DIS
LIN {X 85.3143,Y -15.8843,Z 85,A -16.1188,B 24.9172,C -2.1017,E1 25.1568,E2 461.0554} C_DIS
LIN {X 84.6719,Y -19.0137,Z 85,A -18.2136,B 24.9176,C -2.0955,E1 25.1556,E2 463.1526} C_DIS
LIN {X 83.9146,Y -22.1174,Z 85,A -20.3082,B 24.9181,C -2.0894,E1 25.1541,E2 465.2495} C_DIS
LIN {X 83.0437,Y -25.191,Z 85,A -22.4032,B 24.9186,C -2.0833,E1 25.1525,E2 467.347} C_DIS
LIN {X 82.0602,Y -28.2306,Z 85,A -24.4982,B 24.9191,C -2.0772,E1 25.1506,E2 469.4444} C_DIS
LIN {X 80.9655,Y -31.2318,Z 85,A -26.5932,B 24.9196,C -2.0712,E1 25.1485,E2 471.5419} C_DIS
LIN {X 79.7611,Y -34.1908,Z 85,A -28.6887,B 24.92,C -2.0653,E1 25.1463,E2 473.6399} C_DIS
LIN {X 78.4486,Y -37.1034,Z 85,A -30.7694,B 24.9204,C -2.06,E1 25.1438,E2 475.7219} C_DIS
LIN {X 77.0298,Y -39.9657,Z 85,A -32.8798,B 24.9209,C -2.0537,E1 25.1412,E2 477.8359} C_DIS
LIN {X 75.5065,Y -42.7739,Z 85,A -34.9759,B 24.9213,C -2.048,E1 25.1383,E2 479.9345} C_DIS
LIN {X 73.881,Y -45.5241,Z 85,A -37.072,B 24.9218,C -2.0425,E1 25.1353,E2 482.033} C_DIS
LIN {X 72.1553,Y -48.2126,Z 85,A -39.1686,B 24.9222,C -2.037,E1 25.1321,E2 484.132} C_DIS
LIN {X 70.3318,Y -50.8358,Z 85,A -41.2652,B 24.9226,C -2.0316,E1 25.1287,E2 486.231} C_DIS
LIN {X 68.413,Y -53.3901,Z 85,A -43.3474,B 24.923,C -2.0269,E1 25.1251,E2 488.3145} C_DIS
LIN {X 66.4016,Y -55.872,Z 85,A -45.4446,B 24.9233,C -2.0218,E1 25.1214,E2 490.4141} C_DIS
LIN {X 64.3001,Y -58.2782,Z 85,A -47.557,B 24.9238,C -2.0164,E1 25.1175,E2 492.5299} C_DIS
LIN {X 62.1114,Y -60.6054,Z 85,A -49.6549,B 24.9241,C -2.0116,E1 25.1134,E2 494.6302} C_DIS
LIN {X 59.8386,Y -62.8505,Z 85,A -51.7385,B 24.9244,C -2.0074,E1 25.1092,E2 496.7149} C_DIS
LIN {X 57.4847,Y -65.0104,Z 85,A -53.852,B 24.9248,C -2.0024,E1 25.1048,E2 498.8318} C_DIS
LIN {X 55.0529,Y -67.0822,Z 85,A -55.9362,B 24.9251,C -1.9985,E1 25.1004,E2 500.917} C_DIS
LIN {X 52.5465,Y -69.0631,Z 85,A -58.0355,B 24.9254,C -1.9944,E1 25.0957,E2 503.0185} C_DIS
LIN {X 50.0307,Y -70.9063,Z 85,A -60.0922,B 24.9257,C -1.9902,E1 25.0911,E2 505.0778} C_DIS
LIN {X 47.3235,Y -72.7415,Z 85,A -62.2358,B 24.926,C -1.9865,E1 25.0861,E2 507.223} C_DIS
LIN {X 44.6141,Y -74.4341,Z 85,A -64.3363,B 24.9263,C -1.9829,E1 25.0811,E2 509.3256} C_DIS
LIN {X 41.8441,Y -76.0257,Z 85,A -66.4525,B 24.9266,C -1.9789,E1 25.0759,E2 511.4448} C_DIS
LIN {X 39.0175,Y -77.5144,Z 85,A -68.5541,B 24.9268,C -1.9757,E1 25.0707,E2 513.5484} C_DIS
LIN {X 36.1379,Y -78.898,Z 85,A -70.6412,B 24.927,C -1.9731,E1 25.0654,E2 515.6362} C_DIS
LIN {X 33.2094,Y -80.1747,Z 85,A -72.7588,B 24.9273,C -1.9697,E1 25.0599,E2 517.7567} C_DIS
LIN {X 30.2359,Y -81.3427,Z 85,A -74.862,B 24.9275,C -1.9671,E1 25.0544,E2 519.8616} C_DIS
LIN {X 27.2214,Y -82.4005,Z 85,A -76.9655,B 24.9276,C -1.9646,E1 25.0489,E2 521.9668} C_DIS
LIN {X 24.1701,Y -83.3466,Z 85,A -79.0695,B 24.9278,C -1.9624,E1 25.0432,E2 524.0724} C_DIS
LIN {X 21.0859,Y -84.1797,Z 85,A -81.1741,B 24.9279,C -1.9604,E1 25.0376,E2 526.1785} C_DIS
LIN {X 17.9732,Y -84.8988,Z 85,A -83.2643,B 24.928,C -1.9591,E1 25.0319,E2 528.2691} C_DIS
LIN {X 14.8361,Y -85.5028,Z 85,A -85.3849,B 24.9282,C -1.957,E1 25.026,E2 530.3922} C_DIS
LIN {X 11.679,Y -85.991,Z 85,A -87.4723,B 24.9282,C -1.9563,E1 25.0203,E2 532.4795} C_DIS
LIN {X 8.506,Y -86.3626,Z 85,A -89.5978,B 24.9284,C -1.9546,E1 25.0143,E2 534.6077} C_DIS
LIN {X 5.3214,Y -86.6171,Z 85,A -91.6904,B 24.9284,C -1.9541,E1 25.0085,E2 536.7002} C_DIS
LIN {X 2.1297,Y -86.7543,Z 85,A -93.7981,B 24.9284,C -1.9535,E1 25.0026,E2 538.8091} C_DIS
LIN {X 2.1297,Y -86.7543,Z 85,A -93.7981,B 24.9284,C -1.9535,E1 25.0026,E2 538.8091} C_DIS
Enddeposition()
LIN {X 0.5636,Y -85.8504,Z 85,A -93.432,B 24.924,C -2.0139,E1 25.0041,E2 538.2998} C_DIS
Startdeposition()
$VEL.CP = VEL_PRINT
LIN {X 5.0289,Y -85.7107,Z 85,A -90.7819,B 24.9247,C -2.0042,E1 25.0114,E2 535.6733} C_DIS
LIN {X 9.9955,Y -85.2738,Z 85,A -87.9022,B 24.9256,C -1.9917,E1 25.0193,E2 532.8251} C_DIS
LIN {X 15.5328,Y -84.4416,Z 85,A -84.0011,B 24.925,C -1.9996,E1 25.0301,E2 528.9091} C_DIS
LIN {X 17.9112,Y -83.9695,Z 85,A -82.225,B 24.9245,C -2.0061,E1 25.035,E2 527.1198} C_DIS
LIN {X 21.0028,Y -83.25,Z 85,A -79.9906,B 24.9241,C -2.0119,E1 25.0411,E2 524.8748} C_DIS
LIN {X 24.6172,Y -82.2531,Z 85,A -77.5516,B 24.9241,C -2.0126,E1 25.0476,E2 522.4382} C_DIS
LIN {X 27.8348,Y -81.2215,Z 85,A -75.2603,B 24.9237,C -2.0166,E1 25.0537,E2 520.1419} C_DIS
LIN {X 30.9927,Y -80.0698,Z 85,A -73.0353,B 24.9236,C -2.019,E1 25.0595,E2 517.9159} C_DIS
LIN {X 34.0922,Y -78.7992,Z 85,A -70.8444,B 24.9234,C -2.0208,E1 25.0652,E2 515.726} C_DIS
LIN {X 36.804,Y -77.5704,Z 85,A -68.7829,B 24.923,C -2.0263,E1 25.0704,E2 513.6567} C_DIS
LIN {X 39.7564,Y -76.0989,Z 85,A -65.8919,B 24.9209,C -2.0532,E1 25.0777,E2 510.7102} C_DIS
LIN {X 43.3996,Y -74.0818,Z 85,A -63.8909,B 24.9226,C -2.032,E1 25.0824,E2 508.7653} C_DIS
LIN {X 46.0942,Y -72.436,Z 85,A -61.8041,B 24.9223,C -2.0353,E1 25.0873,E2 506.6775} C_DIS
LIN {X 48.8883,Y -70.5796,Z 85,A -59.3826,B 24.9215,C -2.0459,E1 25.093,E2 504.239} C_DIS
LIN {X 52.0346,Y -68.2946,Z 85,A -56.8853,B 24.9213,C -2.048,E1 25.0986,E2 501.7456} C_DIS
LIN {X 54.7828,Y -66.109,Z 85,A -54.7207,B 24.9214,C -2.0471,E1 25.1032,E2 499.5914} C_DIS
LIN {X 57.0546,Y -64.159,Z 85,A -52.8133,B 24.9214,C -2.0486,E1 25.1072,E2 497.688} C_DIS
LIN {X 59.045,Y -62.3323,Z 85,A -50.7808,B 24.9204,C -2.0606,E1 25.1114,E2 495.6354} C_DIS
LIN {X 61.5082,Y -59.9038,Z 85,A -48.4873,B 24.92,C -2.0657,E1 25.1159,E2 493.3396} C_DIS
LIN {X 63.8491,Y -57.4008,Z 85,A -46.3622,B 24.92,C -2.0659,E1 25.1199,E2 491.2234} C_DIS
LIN {X 65.3113,Y -55.7313,Z 85,A -44.7841,B 24.9194,C -2.0731,E1 25.1228,E2 489.6356} C_DIS
LIN {X 68.4784,Y -51.7911,Z 85,A -41.4534,B 24.9188,C -2.0805,E1 25.1286,E2 486.3029} C_DIS
LIN {X 70.5537,Y -48.9256,Z 85,A -39.097,B 24.9183,C -2.0868,E1 25.1324,E2 483.9431} C_DIS
LIN {X 72.3539,Y -46.222,Z 85,A -37.2103,B 24.9186,C -2.0832,E1 25.1352,E2 482.0743} C_DIS
LIN {X 74.7785,Y -42.1883,Z 85,A -33.9045,B 24.9175,C -2.0979,E1 25.14,E2 478.7509} C_DIS
LIN {X 76.1509,Y -39.6577,Z 85,A -32.1326,B 24.9175,C -2.0984,E1 25.1423,E2 476.9871} C_DIS
LIN {X 77.3755,Y -37.2098,Z 85,A -30.149,B 24.9166,C -2.1092,E1 25.1447,E2 474.9885} C_DIS
LIN {X 78.7746,Y -34.1485,Z 85,A -27.9086,B 24.916,C -2.1158,E1 25.1473,E2 472.7449} C_DIS
LIN {X 80.024,Y -31.1092,Z 85,A -25.7089,B 24.9155,C -2.1227,E1 25.1496,E2 470.5411} C_DIS
LIN {X 81.1652,Y -27.9989,Z 85,A -23.4734,B 24.9149,C -2.1303,E1 25.1516,E2 468.3} C_DIS
LIN {X 81.963,Y -25.5659,Z 85,A -21.8022,B 24.9146,C -2.1344,E1 25.1531,E2 466.6287} C_DIS
LIN {X 83.0502,Y -21.7801,Z 85,A -19.2067,B 24.914,C -2.1415,E1 25.155,E2 464.0314} C_DIS
LIN {X 83.7515,Y -18.9053,Z 85,A -17.1758,B 24.9133,C -2.1497,E1 25.1563,E2 461.9929} C_DIS
LIN {X 84.3062,Y -16.2479,Z 85,A -14.5745,B 24.9106,C -2.1831,E1 25.1577,E2 459.328} C_DIS
LIN {X 85.0449,Y -11.7874,Z 85,A -12.5142,B 24.9126,C -2.1592,E1 25.1585,E2 457.3362} C_DIS
LIN {X 85.6281,Y -6.2938,Z 85,A -8.7106,B 24.9113,C -2.175,E1 25.1595,E2 453.5178} C_DIS
LIN {X 85.8146,Y -2.7208,Z 85,A -6.437,B 24.911,C -2.1787,E1 25.1597,E2 451.249} C_DIS
LIN {X 85.8596,Y 0.0044,Z 85,A -3.5177,B 24.9073,C -2.223,E1 25.1597,E2 448.2424} C_DIS
LIN {X 85.7006,Y 5.2118,Z 85,A -0.3759,B 24.9073,C -2.2223,E1 25.1592,E2 445.1211} C_DIS
LIN {X 85.3408,Y 9.4189,Z 85,A 1.6894,B 24.9088,C -2.2049,E1 25.1586,E2 443.109} C_DIS
LIN {X 84.8846,Y 12.8915,Z 85,A 3.9674,B 24.9084,C -2.2102,E1 25.1577,E2 440.832} C_DIS
LIN {X 84.3229,Y 16.1614,Z 85,A 6.1926,B 24.9078,C -2.2175,E1 25.1566,E2 438.6027} C_DIS
LIN {X 83.6271,Y 19.4435,Z 85,A 8.3279,B 24.9075,C -2.2208,E1 25.1553,E2 436.472} C_DIS
LIN {X 82.9109,Y 22.3009,Z 85,A 10.3626,B 24.9068,C -2.2291,E1 25.1539,E2 434.4292} C_DIS
LIN {X 82.0138,Y 25.4021,Z 85,A 12.4887,B 24.9063,C -2.2346,E1 25.1522,E2 432.3023} C_DIS
LIN {X 81.1749,Y 27.9716,Z 85,A 14.2303,B 24.9061,C -2.2378,E1 25.1506,E2 430.5631} C_DIS
LIN {X 80.2867,Y 30.4233,Z 85,A 16.9363,B 24.9028,C -2.2762,E1 25.1478,E2 427.7812} C_DIS
LIN {X 78.4746,Y 34.8353,Z 85,A 19.0945,B 24.905,C -2.2499,E1 25.1455,E2 425.697} C_DIS
LIN {X 76.5207,Y 38.9376,Z 85,A 22.1884,B 24.9041,C -2.2604,E1 25.1417,E2 422.5949} C_DIS
LIN {X 74.9824,Y 41.8232,Z 85,A 24.2349,B 24.9041,C -2.2617,E1 25.139,E2 420.5561} C_DIS
LIN {X 73.2485,Y 44.7911,Z 85,A 27.6564,B 24.9002,C -2.3063,E1 25.1339,E2 417.0466} C_DIS
LIN {X 70.5122,Y 48.9854,Z 85,A 29.8543,B 24.9028,C -2.2757,E1 25.1306,E2 414.932} C_DIS
LIN {X 68.7693,Y 51.4039,Z 85,A 31.9525,B 24.9021,C -2.2842,E1 25.1271,E2 412.8236} C_DIS
LIN {X 66.5269,Y 54.2751,Z 85,A 34.3892,B 24.9016,C -2.2902,E1 25.1228,E2 410.3842} C_DIS
LIN {X 64.2403,Y 56.9639,Z 85,A 36.6299,B 24.9015,C -2.2917,E1 25.1188,E2 408.1501} C_DIS
LIN {X 62.0898,Y 59.3005,Z 85,A 38.7294,B 24.9011,C -2.2957,E1 25.1147,E2 406.0504} C_DIS
LIN {X 59.7837,Y 61.624,Z 85,A 40.9064,B 24.9007,C -2.3,E1 25.1104,E2 403.8722} C_DIS
LIN {X 57.4626,Y 63.7938,Z 85,A 43.1005,B 24.9002,C -2.3067,E1 25.1059,E2 401.6711} C_DIS
LIN {X 54.7488,Y 66.1372,Z 85,A 45.2467,B 24.9005,C -2.3031,E1 25.1014,E2 399.5417} C_DIS
LIN {X 51.4295,Y 68.7501,Z 85,A 48.7196,B 24.8982,C -2.3298,E1 25.0936,E2 396.0185} C_DIS
LIN {X 47.4926,Y 71.5267,Z 85,A 51.4373,B 24.8991,C -2.3186,E1 25.0874,E2 393.3364} C_DIS
LIN {X 44.828,Y 73.2261,Z 85,A 53.5671,B 24.8988,C -2.3225,E1 25.0823,E2 391.2042} C_DIS
LIN {X 41.9945,Y 74.8867,Z 85,A 55.5333,B 24.8992,C -2.3183,E1 25.0776,E2 389.2539} C_DIS
LIN {X 37.6702,Y 77.1541,Z 85,A 59.7807,B 24.896,C -2.3546,E1 25.0668,E2 384.9321} C_DIS
LIN {X 33.9207,Y 78.8739,Z 85,A 62.0608,B 24.8971,C -2.3422,E1 25.0611,E2 382.6868} C_DIS
LIN {X 30.0353,Y 80.4337,Z 85,A 64.564,B 24.8976,C -2.3356,E1 25.0546,E2 380.2049} C_DIS
LIN {X 26.8158,Y 81.5635,Z 85,A 66.754,B 24.8977,C -2.3347,E1 25.0488,E2 378.0212} C_DIS
LIN {X 23.8037,Y 82.4929,Z 85,A 68.8681,B 24.8976,C -2.3366,E1 25.0432,E2 375.9065} C_DIS
LIN {X 20.7219,Y 83.3204,Z 85,A 71.0467,B 24.8973,C -2.3394,E1 25.0373,E2 373.7244} C_DIS
LIN {X 17.6294,Y 84.029,Z 85,A 73.1042,B 24.8973,C -2.3386,E1 25.0317,E2 371.6716} C_DIS
LIN {X 14.44,Y 84.6351,Z 85,A 75.3554,B 24.8971,C -2.342,E1 25.0255,E2 369.4147} C_DIS
LIN {X 10.7589,Y 85.1813,Z 85,A 77.6893,B 24.8974,C -2.338,E1 25.0191,E2 367.0924} C_DIS
LIN {X 7.6518,Y 85.5163,Z 85,A 80.183,B 24.8963,C -2.351,E1 25.0121,E2 364.5694} C_DIS
LIN {X 3.0399,Y 85.8048,Z 85,A 83.2791,B 24.8963,C -2.3512,E1 25.0034,E2 361.4738} C_DIS
LIN {X -3.1263,Y 85.8021,Z 85,A 88.2154,B 24.8941,C -2.3757,E1 24.9895,E2 356.4788} C_DIS
LIN {X -8.3806,Y 85.449,Z 85,A 90.7012,B 24.8971,C -2.3422,E1 24.9828,E2 354.0714} C_DIS
LIN {X -11.632,Y 85.0672,Z 85,A 92.5632,B 24.898,C -2.3311,E1 24.9777,E2 352.2345} C_DIS
LIN {X -14.5457,Y 84.6174,Z 85,A 94.8347,B 24.8974,C -2.3389,E1 24.9714,E2 349.9423} C_DIS
LIN {X -18.0574,Y 83.9376,Z 85,A 97.1541,B 24.8977,C -2.3349,E1 24.965,E2 347.6297} C_DIS
LIN {X -21.3755,Y 83.1542,Z 85,A 99.4744,B 24.8977,C -2.3341,E1 24.9588,E2 345.3081} C_DIS
LIN {X -25.1854,Y 82.081,Z 85,A 101.9724,B 24.8984,C -2.3269,E1 24.9521,E2 342.823} C_DIS
LIN {X -28.8132,Y 80.8795,Z 85,A 104.6004,B 24.8984,C -2.3261,E1 24.9451,E2 340.1919} C_DIS
LIN {X -31.73,Y 79.7802,Z 85,A 106.723,B 24.8986,C -2.3246,E1 24.9396,E2 338.0683} C_DIS
LIN {X -34.616,Y 78.5708,Z 85,A 108.6636,B 24.8993,C -2.3173,E1 24.9347,E2 336.1407} C_DIS
LIN {X -37.437,Y 77.2663,Z 85,A 110.9104,B 24.8991,C -2.3191,E1 24.929,E2 333.8837} C_DIS
LIN {X -40.4949,Y 75.7094,Z 85,A 113.277,B 24.8992,C -2.3176,E1 24.9231,E2 331.5143} C_DIS
LIN {X -43.2386,Y 74.177,Z 85,A 115.3918,B 24.8995,C -2.3144,E1 24.918,E2 329.4008} C_DIS
LIN {X -46.2801,Y 72.3166,Z 85,A 117.7192,B 24.9,C -2.3085,E1 24.9125,E2 327.0802} C_DIS
LIN {X -48.6706,Y 70.731,Z 85,A 119.5997,B 24.9004,C -2.3038,E1 24.9082,E2 325.2046} C_DIS
LIN {X -53.4571,Y 67.1859,Z 85,A 123.4027,B 24.9016,C -2.2905,E1 24.8997,E2 321.4195} C_DIS
LIN {X -56.7976,Y 64.3874,Z 85,A 126.5901,B 24.9014,C -2.2921,E1 24.8929,E2 318.2161} C_DIS
LIN {X -60.0836,Y 61.3308,Z 85,A 129.701,B 24.9018,C -2.2884,E1 24.8866,E2 315.1012} C_DIS
LIN {X -63.019,Y 58.3089,Z 85,A 132.7833,B 24.9017,C -2.2893,E1 24.8807,E2 312.0033} C_DIS
Enddeposition()
END
